	// WX2A ROT
IF WX2TargetPos.nRotPos + WX2TargetPos.nRotCatch > WX^.Rot_A.Out.DistancePos_PO AND
	WX2TargetPos.nRotPos - WX2TargetPos.nRotCatch < WX^.Rot_A.Out.DistancePos_PO THEN
		WX^.Rot_A.bStopMove := TRUE;
END_IF

	// WX2A CLAMP
IF WX2TargetPos.nClampPos + WX2TargetPos.nClampCatch > WX^.Clamp_A.Out.DistancePos_PO AND
	WX2TargetPos.nClampPos - WX2TargetPos.nClampCatch < WX^.Clamp_A.Out.DistancePos_PO THEN
		WX^.Clamp_A.bStopMove := TRUE;
END_IF

	// WX2B VERT
IF WX2TargetPos.nVertPos + WX2TargetPos.nVertCatch > WX^.Vert_B.Out.DistancePos_PO AND
	WX2TargetPos.nVertPos - WX2TargetPos.nVertCatch < WX^.Vert_B.Out.DistancePos_PO THEN
		WX^.Vert_B.bStopMove := TRUE;
END_IF

	// WX2B ROT
IF WX2TargetPos.nRotPos + WX2TargetPos.nRotCatch > WX^.Rot_B.Out.DistancePos_PO AND
	WX2TargetPos.nRotPos - WX2TargetPos.nRotCatch < WX^.Rot_B.Out.DistancePos_PO THEN
		WX^.Rot_B.bStopMove := TRUE;
END_IF

	// WX2B CLAMP
IF WX2TargetPos.nClampPos + WX2TargetPos.nClampCatch > WX^.Clamp_B.Out.DistancePos_PO AND
	WX2TargetPos.nClampPos - WX2TargetPos.nClampCatch < WX^.Clamp_B.Out.DistancePos_PO THEN
		WX^.Clamp_B.bStopMove := TRUE;
END_IF




	// This is to give the axes time to stop, before we move onto the next step
IF WX^.Vert_A.StopCase = 100 AND WX^.Rot_A.StopCase = 100 AND WX^.Clamp_A.StopCase = 100 AND
	WX^.Vert_B.StopCase = 100 AND WX^.Rot_B.StopCase = 100 AND WX^.Clamp_B.StopCase = 100 THEN
	bInPosition := TRUE;
ELSE
	bInPosition := FALSE;
END_IF

IF bClamped THEN
	IF WX^.Vert_A.StopCase = 100 AND WX^.Rot_A.StopCase = 100 AND WX^.Vert_B.StopCase = 100 THEN
		bInPosition := TRUE;
	ELSE
		bInPosition := FALSE;
	END_IF
END_IF

armsInTargetPosition := bInPosition;
END_METHOD

METHOD CleanUpMove : BOOL
(*
	This method assumes that the movement from the initial 'big' move has ended.
*)
IF NOT bInitCleanUpTrigger THEN
	enableAltSpeed();
	
		// Reload Target Position into our ClearpathPositionABS
	WX^.VertDisReq_PI 	:= REAL_TO_INT(WX2TargetPos.nVertPos);
	WX^.RotDegReq_PI  	:= REAL_TO_INT(WX2TargetPos.nRotPos);
	WX^.ClampDisReq_PI := REAL_TO_INT(WX2TargetPos.nClampPos);
	
		// If we are clamped, we don't move all axis
	IF NOT bClamped THEN
		WX^.bPresetMoveTrigger := TRUE;
	ELSE
		WX^.Vert_A.bPresetMoveTrigger := TRUE;
		WX^.Vert_B.bPresetMoveTrigger := TRUE;
		WX^.Rot_A.bPresetMoveTrigger  := TRUE;
			
		WX^.Vert_A.bMove_PI := TRUE;
		WX^.Vert_B.bMove_PI := TRUE;
		WX^.Rot_A.bMove_PI  := TRUE;
	END_IF
	
	enableAltSpeed();
	
	bInitCleanUpTrigger     := TRUE;
END_IF

enableAltSpeed();

CleanUpMove := precisionMoveChecker();
END_METHOD

METHOD disableAltSpeed : BOOL
VAR
	bDetect : BOOL := FALSE;
END_VAR

(* 
	This method returns TRUE if  alt speed control was DISABLED already.
*)
bDetect := FALSE;

IF NOT WX^.Vert_A.bAltSpeedControl OR NOT WX^.Vert_B.bAltSpeedControl  THEN
	bDetect := TRUE;
END_IF

IF NOT WX^.Rot_A.bAltSpeedControl OR NOT WX^.Rot_B.bAltSpeedControl THEN
	bDetect := TRUE;
END_IF

IF NOT WX^.Clamp_A.bAltSpeedControl OR NOT WX^.Clamp_A.bAltSpeedControl THEN
	bDetect := TRUE;
END_IF

WX^. Vert_A.bAltSpeedControl := FALSE;
WX^.  Rot_A.bAltSpeedControl := FALSE;
WX^.Clamp_A.bAltSpeedControl := FALSE;

WX^. Vert_B.bAltSpeedControl := FALSE;
WX^.  Rot_B.bAltSpeedControl := FALSE;
WX^.Clamp_A.bAltSpeedControl := FALSE;

disableAltSpeed := bDetect;
END_METHOD

METHOD enableAltSpeed : BOOL
VAR
	bDetect : BOOL := FALSE;
END_VAR
(* 
	This method returns TRUE if  alt speed control was ENABLED already.
*)
bDetect := FALSE;

IF WX^.Vert_A.bAltSpeedControl OR WX^.Vert_B.bAltSpeedControl  THEN
	bDetect := TRUE;
END_IF

IF WX^.Rot_A.bAltSpeedControl OR WX^. Rot_B.bAltSpeedControl THEN
	bDetect := TRUE;
END_IF

IF WX^.Clamp_A.bAltSpeedControl OR WX^.Clamp_B.bAltSpeedControl THEN
	bDetect := TRUE;
END_IF

WX^. Vert_A.bAltSpeedControl := TRUE;
WX^.  Rot_A.bAltSpeedControl := TRUE;
WX^.Clamp_A.bAltSpeedControl := TRUE;

WX^. Vert_B.bAltSpeedControl := TRUE;
WX^.  Rot_B.bAltSpeedControl := TRUE;
WX^.Clamp_B.bAltSpeedControl := TRUE;

enableAltSpeed := bDetect;
END_METHOD

METHOD MoveArms : BOOL
VAR_INPUT
	position : sBogieArmPosition;
END_VAR
(*
	Author @ Joseph Barton	

	This method is initiating and monitoring the initial move for a preset move command.
*)

	// If we are not busy moving somewhere.
IF NOT bBusy THEN	
	bBusy 		  := TRUE;	// We are now busy.
	bMoveComplete := FALSE;	// And our move is not complete.
							// 	If we are already in the target position,
							// 	That will be determined later in this cycle.
	tStartTime := TIME(); 	// Save the start time, for the timeout error tracking.
							
		// This is the 'big' move, so we disable altenate speed to move quickly
	disableAltSpeed();		
	
		// set our target position for position checking.
	WX2TargetPos := position;	
	
		// Tell the Auto-movement part of our clearpath library our desired location.
	WX^.VertDisReq_PI 	:= REAL_TO_INT(WX2TargetPos.nVertPos); 	
	WX^.RotDegReq_PI  	:= REAL_TO_INT(WX2TargetPos.nRotPos);
	WX^.ClampDisReq_PI := REAL_TO_INT(WX2TargetPos.nClampPos);
	
		// IF we are NOT clamped we can use the bPresetMoveTrigger boolean to
		//		give the library the right information on how te move.
	IF NOT bClamped THEN
		WX^.bPresetMoveTrigger := TRUE;
	ELSE
		
			// If we are clamped, then we cannot move all 6 motors,
			//		and we have to manually tell our desired axis
			//		that we are moving them to a preset position.
		WX^.Vert_A.bPresetMoveTrigger := TRUE;
		WX^.Vert_B.bPresetMoveTrigger := TRUE;
		WX^.Rot_A.bPresetMoveTrigger  := TRUE;
		
			// Then tell them to move.
		WX^.Vert_A.bMove_PI := TRUE;
		WX^.Vert_B.bMove_PI := TRUE;
		WX^.Rot_A.bMove_PI  := TRUE;
	END_IF
	
	disableAltSpeed();
END_IF

	// disableing alternate speed each cycle is too much,
	//		but there is a glitch where it will go into
	// 		alternate speed 'randomly'. I will have to
	//		fix it soon.
disableAltSpeed();

	// Check if we are in the correct position each cycle.
MoveArms := armsInTargetPosition();
END_METHOD

METHOD partPresent : BOOL
VAR_INPUT
END_VAR

(* 
	This method returns true if there is a part detected by the part present sensor.
	
	This still needs to be implemented, but because the Part Present Sensors do not exist yet, this is what we got.
*)
partPresent := FALSE;
END_METHOD

METHOD precisionMoveChecker : BOOL
VAR
	bWX2AVertInLocation  : BOOL := FALSE;
	bWX2ARotInLocation   : BOOL := FALSE;
	bWX2AClampInLocation : BOOL := FALSE;
	
	bWX2BVertInLocation  : BOOL := FALSE;
	bWX2BRotInLocation 	 : BOOL := FALSE;
	bWX2BClampInLocation : BOOL := FALSE;
END_VAR
	// Vert_A
IF WX2TargetPos.nVertPos + WX2TargetPos.nVertTolerance > WX^.Vert_A.Out.DistancePos_PO AND
 	WX2TargetPos.nVertPos - WX2TargetPos.nVertTolerance < WX^.Vert_A.Out.DistancePos_PO THEN
		bWX2AVertInLocation := TRUE;
		WX^.Vert_A.bStopMove := TRUE;
ELSE
	WX^.Vert_A.bStopMove := FALSE;
END_IF
	
	// Rot_A
IF WX2TargetPos.nRotPos + WX2TargetPos.nRotTolerance > WX^.Rot_A.Out.DistancePos_PO AND
	WX2TargetPos.nRotPos - WX2TargetPos.nRotTolerance < WX^.Rot_A.Out.DistancePos_PO THEN
		bWX2ARotInLocation := TRUE;
		WX^.Rot_A.bStopMove := TRUE;
ELSE
	WX^.Rot_A.bStopMove := FALSE;
END_IF

	// Clamp_A
IF WX2TargetPos.nClampPos + WX2TargetPos.nClampTolerance > WX^.Clamp_A.Out.DistancePos_PO AND
	WX2TargetPos.nClampPos - WX2TargetPos.nClampTolerance < WX^.Clamp_A.Out.DistancePos_PO THEN
		bWX2AClampInLocation := TRUE;
		WX^.Clamp_A.bStopMove := TRUE;
ELSE
	WX^.Clamp_A.bStopMove := FALSE;
END_IF

	// Vert_B
IF WX2TargetPos.nVertPos + WX2TargetPos.nVertTolerance > WX^.Vert_B.Out.DistancePos_PO AND
 	WX2TargetPos.nVertPos - WX2TargetPos.nVertTolerance < WX^.Vert_B.Out.DistancePos_PO THEN
		bWX2BVertInLocation := TRUE;
		WX^.Vert_B.bStopMove := TRUE;
ELSE
	WX^.Vert_B.bStopMove := FALSE;
END_IF
	
	// Rot_B
IF WX2TargetPos.nRotPos + WX2TargetPos.nRotTolerance > WX^.Rot_B.Out.DistancePos_PO AND
	WX2TargetPos.nRotPos - WX2TargetPos.nRotTolerance < WX^.Rot_B.Out.DistancePos_PO THEN
		bWX2BRotInLocation := TRUE;
		WX^.Rot_B.bStopMove := TRUE;
ELSE
	WX^.Rot_B.bStopMove := FALSE;
END_IF

	// Clamp_B
IF WX2TargetPos.nClampPos + WX2TargetPos.nClampTolerance > WX^.Clamp_B.Out.DistancePos_PO AND
	WX2TargetPos.nClampPos - WX2TargetPos.nClampTolerance < WX^.Clamp_B.Out.DistancePos_PO THEN
		bWX2BClampInLocation := TRUE;
		WX^.Clamp_B.bStopMove := TRUE;
ELSE
	WX^.Clamp_B.bStopMove := FALSE;
END_IF

	// Check if all axis are in location, and return TRUE; ELSE return FALSE;
IF bWX2AVertInLocation AND bWX2ARotInLocation AND bWX2AClampInLocation AND
	bWX2BVertInLocation AND bWX2BRotInLocation AND bWX2BClampInLocation THEN
		
		WX^.Clamp_B.bStopMove := FALSE;
		WX^.Rot_B.bStopMove := FALSE;
		WX^.Vert_B.bStopMove := FALSE;
		WX^.Clamp_A.bStopMove := FALSE;
		WX^.Rot_A.bStopMove := FALSE;
		WX^.Vert_A.bStopMove := FALSE;
		
		precisionMoveChecker := TRUE;
	
ELSE
	precisionMoveChecker := FALSE;
END_IF

	// IF we are clamped then we are checking for the Vert_A, Vert_B, & Rot_A axis only.
IF bClamped THEN
	IF bWX2AVertInLocation AND bWX2ARotInLocation AND bWX2BVertInLocation THEN
		
		WX^.Vert_B.bStopMove := FALSE;
		WX^.Rot_A.bStopMove := FALSE;
		WX^.Vert_A.bStopMove := FALSE;
		
		precisionMoveChecker := TRUE;
	END_IF
END_IF
END_METHOD

ACTION startAllMovement:
WX^.Vert_A.bStopMove 	:= FALSE;
WX^.Rot_A.bStopMove 	:= FALSE;
WX^.Clamp_A.bStopMove 	:= FALSE;
WX^.Vert_B.bStopMove 	:= FALSE;
WX^.Rot_B.bStopMove  	:= FALSE;
WX^.Clamp_B.bStopMove 	:= FALSE;
END_ACTION

ACTION stopAllMovement:
WX^.Vert_A.bStopMove 	:= TRUE;
WX^.Rot_A.bStopMove 	:= TRUE;
WX^.Clamp_A.bStopMove 	:= TRUE;
WX^.Vert_B.bStopMove 	:= TRUE;
WX^.Rot_B.bStopMove 	:= TRUE;
WX^.Clamp_B.bStopMove 	:= TRUE;
END_ACTION

END_FUNCTION_BLOCK

// ---- Machine System/FUNCTIONS/F_PartIsPresent.TcPOU
FUNCTION F_PartIsPresent : BOOL
VAR_INPUT
	WX : sBogie;
END_VAR
VAR
END_VAR

IF (WX.A.bPP1_Input AND WX.A.bPP2_Input AND WX.B.bPP1_Input AND WX.A.bPP2_Input) OR NOT(WX.bEnabled) THEN
	F_PartIsPresent := 1;
	ELSE
		F_PartIsPresent := 0;
END_IF

END_FUNCTION

// ---- Machine System/FUNCTIONS/F_PartIsPresentAndClamped.TcPOU
FUNCTION F_PartIsPresentAndClamped : BOOL
VAR_INPUT
	WX : sBogie;
END_VAR
VAR
END_VAR

IF (WX.A.bPP1_Input AND WX.A.bPP2_Input AND WX.B.bPP1_Input AND WX.A.bPP2_Input AND WX.A.bClamped AND WX.B.bClamped) OR NOT(WX.bEnabled) THEN
	F_PartIsPresentAndClamped := 1;
	ELSE
		F_PartIsPresentAndClamped := 0;
END_IF

END_FUNCTION

// ---- Machine System/FUNCTIONS/F_IsEmpty.TcPOU
FUNCTION F_IsEmpty : BOOL
VAR_INPUT
	WX : sBogie;
END_VAR
VAR
END_VAR

IF WX.A.bPP1_Input = 0 AND WX.A.bPP2_Input = 0 AND WX.B.bPP2_Input = 0 AND WX.B.bPP2_Input = 0 THEN
	F_IsEmpty := 1;
	ELSE 
		F_IsEmpty := 0;
END_IF

END_FUNCTION

// ---- Machine System/FUNCTIONS/F_ArmsInLoadOrientation.TcPOU
FUNCTION F_ArmsInLoadOrientation : BOOL
VAR_INPUT
END_VAR
VAR
END_VAR

END_FUNCTION

// ---- Machine System/FUNCTIONS/F_PartPickupSuccess.TcPOU
FUNCTION F_PartPickupSuccess : BOOL
VAR_INPUT
	WX : sBogie;
END_VAR
VAR
END_VAR

IF WX.bEnabled THEN
	IF WX.A.bClamped AND WX.B.bClamped AND F_PartIsPresent(WX) AND WX.ConveyorLoadPos = 0 THEN
		
		F_PartPickupSuccess := 1;
 
	ELSE
		F_PartPickupSuccess := 0;
		RETURN;
	END_IF
	
	RETURN;
	
END_IF

END_FUNCTION

// ---- Machine System/FUNCTIONS/F_CheckMoldData.TcPOU
FUNCTION F_CheckMoldData : BOOL
VAR_INPUT
	MoldID 		: INT;
	WX_Enable	: BOOL;
END_VAR
VAR
END_VAR

//Function to check the database for each file string and check for the file on the system 
IF WX_Enable THEN
	IF MoldID = 0 THEN
		RETURN;
		ELSE
			F_CheckMoldData := 1;
		END_IF
	ELSE
		F_CheckMoldData := 1;
END_IF

END_FUNCTION

// ---- CNC HMI/CNC_HMI_HLI_Added_Code.TcPOU
PROGRAM CNC_HMI_HLI_Added_Code
VAR
Scaler : INT :=10000; //change to a scaling variable when deciding to use inches
mdiTest : STRING;
//EventLogger page Reset
	fbEventlogger : FB_TcEventLogger;
	fbAlarm: FB_TcAlarm;
	fbMessage: FB_TcMessage;
	bAlarm: BOOL;
	bMessage : BOOL;
	bIsInitalized: BOOL;
	bClearAlarm: BOOL;
	bConfirmAlarm: BOOL;
//ch1
	SP1_X : fb_HMI_AX;
	SP1_Y : fb_HMI_AX;
	SP1_Z : fb_HMI_AX;
	SP1_A : fb_HMI_AX;
	SP1_C : fb_HMI_AX;
//ch2
	R1_X	: fb_HMI_AX;
	R1_Y	: fb_HMI_AX;
	R1_Z1	: fb_HMI_AX;
	R1_Z2	: fb_HMI_AX;
	R1_C	: fb_HMI_AX;
	
//axis1
(*
Spray_Axis1 : STRING;
SP1_PCS		: STRING;
SP1_ACS		: STRING;
SP1_cmd		: STRING;
SP1_Min		: STRING;
SP1_Max		: STRING;
//axis2

Spray_Axis2 : STRING;
SP2_PCS		: STRING;
SP2_ACS		: STRING;
SP2_cmd		: STRING;
SP2_Min		: STRING;
SP2_Max		: STRING;
SP2_Feed	: string;
//axis3
Spray_Axis3 : STRING;
SP3_PCS		: STRING;
SP3_ACS		: STRING;
SP3_cmd		: STRING;
SP3_min		: STRING;
SP3_max		: STRING;
//axis4
Spray_Axis4 : STRING;
SP4_PCS		: STRING;
SP4_ACS		: STRING;
SP4_cmd		: STRING;
SP4_min		: STRING;
SP4_max		: STRING;
//axis5
Spray_Axis5 : STRING;
SP5_PCS		: STRING;
SP5_ACS		: STRING;
SP5_cmd		: STRING;
Sp5_min		: STRING;
SP5_Max		: STRING;

//channel 2
//axis1
Roll_Axis1 	: STRING;
R1_PCS		: STRING;
R1_ACS		: STRING;
R1_cmd		: STRING;
R1_Min		: STRING;
R1_Max		: STRING;
//axis2
Roll_Axis2 	: STRING;
R2_PCS		: STRING;
R2_ACS		: STRING;
R2_cmd		: STRING;
//axis3
Roll_Axis3 	: STRING;
R3_PCS		: STRING;
R3_ACS		: STRING;
R3_cmd		: STRING;
//axis4
Roll_Axis4 	: STRING;
R4_PCS		: STRING;
R4_ACS		: STRING;
R4_cmd		: STRING;
//axis5
Roll_Axis5 	: STRING;
R5_PCS		: STRING;
R5_ACS		: STRING;
R5_cmd		: STRING;
//axis6
Roll_Axis6 	: STRING;
R6_PCS		: STRING;
R6_ACS		: STRING;
R6_cmd		: STRING;
*)
//gcode access See PRG 'P_GFuctionMonitor()'

END_VAR


// read gcode buffer
	P_GFunctionMonitor();	//Channel 1 G Code Reader
	//P_GFunctionMonitor_2(); 	//channel 2 G Code Reader
//EventLogger Buttons for reset
//	IF NOT bIsInitalized THEN
//	bIsInitalized := TRUE;
//	fbMessage.CreateEx(TC_Events.MyEvents.Start, 0);
//	fbAlarm.CreateEx(TC_Events.MyEvents.Stop, TRUE, 0);
//	END_IF
//	//Test git
//	IF bMessage THEN
//		bMessage := FALSE;
//		fbMessage.Send(0);
//	END_IF
	
//	IF bAlarm THEN
//		bAlarm := FALSE;
//		fbAlarm.Raise(0);
//	END_IF
	
//	IF bClearAlarm THEN
//		bClearAlarm := FALSE;
//		fbAlarm.Clear(0, TRUE);
//	END_IF
//ch1 fb
	SP1_X(chId:=0,chAx:=0,Scaler:=Scaler);
	SP1_Y(chId:=0,chAx:=1,Scaler:=Scaler);
	SP1_Z(chId:=0,chAx:=2,Scaler:=Scaler);
	SP1_A(chId:=0,chAx:=3,Scaler:=Scaler);
	SP1_C(chId:=0,chAx:=4,Scaler:=Scaler);
//ch2 fb
	R1_X(chId:=1,chAx:=0,Scaler:=Scaler);
	R1_Y(chId:=1,chAx:=1,Scaler:=Scaler);
	R1_Z1(chId:=1,chAx:=2,Scaler:=Scaler);
	R1_Z2(chId:=1,chAx:=3,Scaler:=Scaler);
	R1_C(chId:=1,chAx:=4,Scaler:=Scaler);
	
(*  Method for HMI before FB was added.  Use this if While loop fails
	Spray_Axis1 := gpCh[0]^.bahn_state.coord_r[0].axis_name_r.zeichen;
	SP1_PCS		:= FLOAT_TO_STRING(Dint_to_float(gpCh[0]^.bahn_state.coord_r[0].current_position_r)/Scaler);
	SP1_ACS		:= FLOAT_TO_STRING(Dint_to_float(gpCh[0]^.bahn_state.coord_r[0].acs_position_r)/Scaler);
	SP1_CMD		:= FLOAT_TO_STRING(DINT_TO_FLOAT(gpCh[0]^.bahn_state.coord_r[0].cmd_position_r)/Scaler);
	SP1_Min 	:= FLOAT_TO_STRING(DINT_TO_FLOAT(gpAx[0]^.lr_state.conf_neg_software_limit_r)/Scaler);
	SP1_Max 	:= FLOAT_TO_STRING(DINT_TO_FLOAT(gpAx[0]^.lr_state.conf_pos_software_limit_r)/Scaler);
	Spray_Axis2 := gpCh[0]^.bahn_state.coord_r[1].axis_name_r.zeichen;
	SP2_PCS		:= FLOAT_TO_STRING(Dint_to_float(gpCh[0]^.bahn_state.coord_r[1].current_position_r)/Scaler);
	SP2_ACS		:= FLOAT_TO_STRING(Dint_to_float(gpCh[0]^.bahn_state.coord_r[1].acs_position_r)/Scaler);
	SP2_CMD		:= FLOAT_TO_STRING(DINT_TO_FLOAT(gpCh[0]^.bahn_state.coord_r[1].cmd_position_r)/Scaler);
	SP2_Min 	:= FLOAT_TO_STRING(DINT_TO_FLOAT(gpAx[1]^.lr_state.conf_neg_software_limit_r)/Scaler);
	SP2_Max 	:= FLOAT_TO_STRING(DINT_TO_FLOAT(gpAx[1]^.lr_state.conf_pos_software_limit_r)/Scaler);
	SP2_Feed	:= DINT_TO_STRING(gpch[0]^.bahn_state.coord_r[1].w0_velocity_r);
	
	Spray_Axis3 := gpCh[0]^.bahn_state.coord_r[2].axis_name_r.zeichen;
	SP3_PCS		:= FLOAT_TO_STRING(Dint_to_float(gpCh[0]^.bahn_state.coord_r[2].current_position_r)/Scaler);
	SP3_ACS		:= FLOAT_TO_STRING(Dint_to_float(gpCh[0]^.bahn_state.coord_r[2].acs_position_r)/Scaler);
	SP3_CMD		:= FLOAT_TO_STRING(DINT_TO_FLOAT(gpCh[0]^.bahn_state.coord_r[2].cmd_position_r)/Scaler);
	SP3_Min 	:= FLOAT_TO_STRING(DINT_TO_FLOAT(gpAx[2]^.lr_state.conf_neg_software_limit_r)/Scaler);
	SP3_Max 	:= FLOAT_TO_STRING(DINT_TO_FLOAT(gpAx[2]^.lr_state.conf_pos_software_limit_r)/Scaler);
	
	Spray_Axis4 := gpCh[0]^.bahn_state.coord_r[3].axis_name_r.zeichen;
	SP4_PCS		:= FLOAT_TO_STRING(Dint_to_float(gpCh[0]^.bahn_state.coord_r[3].current_position_r)/Scaler);
	SP4_ACS		:= FLOAT_TO_STRING(Dint_to_float(gpCh[0]^.bahn_state.coord_r[3].acs_position_r)/Scaler);
	SP4_CMD		:= FLOAT_TO_STRING(DINT_TO_FLOAT(gpCh[0]^.bahn_state.coord_r[3].cmd_position_r)/Scaler);
	SP4_Min 	:= FLOAT_TO_STRING(DINT_TO_FLOAT(gpAx[3]^.lr_state.conf_neg_software_limit_r)/Scaler);
	SP4_Max 	:= FLOAT_TO_STRING(DINT_TO_FLOAT(gpAx[3]^.lr_state.conf_pos_software_limit_r)/Scaler);
	
	Spray_Axis5 := gpCh[0]^.bahn_state.coord_r[4].axis_name_r.zeichen;
	SP5_PCS		:= FLOAT_TO_STRING(Dint_to_float(gpCh[0]^.bahn_state.coord_r[4].current_position_r)/Scaler);
	SP5_ACS		:= FLOAT_TO_STRING(Dint_to_float(gpCh[0]^.bahn_state.coord_r[4].acs_position_r)/Scaler);
	SP5_CMD		:= FLOAT_TO_STRING(DINT_TO_FLOAT(gpCh[0]^.bahn_state.coord_r[4].cmd_position_r)/Scaler);
	SP5_Min 	:= FLOAT_TO_STRING(DINT_TO_FLOAT(gpAx[4]^.lr_state.conf_neg_software_limit_r)/Scaler);
	SP5_Max 	:= FLOAT_TO_STRING(DINT_TO_FLOAT(gpAx[4]^.lr_state.conf_pos_software_limit_r)/Scaler);
	
	//channel2
	Roll_Axis1 	:= gpCh[1]^.bahn_state.coord_r[0].axis_name_r.zeichen;
	R1_PCS		:= FLOAT_TO_STRING(Dint_to_float(gpCh[1]^.bahn_state.coord_r[0].current_position_r)/Scaler);
	R1_ACS		:= FLOAT_TO_STRING(Dint_to_float(gpCh[1]^.bahn_state.coord_r[0].acs_position_r)/Scaler);
	R1_CMD		:= FLOAT_TO_STRING(Dint_to_float(gpCh[1]^.bahn_state.coord_r[0].cmd_position_r)/Scaler);
	R1_Min 		:= FLOAT_TO_STRING(DINT_TO_FLOAT(gpAx[0]^.lr_state.conf_neg_software_limit_r)/Scaler);
	R1_Max 		:= FLOAT_TO_STRING(DINT_TO_FLOAT(gpAx[0]^.lr_state.conf_pos_software_limit_r)/Scaler);
	
	Roll_Axis2 	:= gpCh[1]^.bahn_state.coord_r[1].axis_name_r.zeichen;
	R2_PCS		:= FLOAT_TO_STRING(Dint_to_float(gpCh[1]^.bahn_state.coord_r[1].current_position_r)/Scaler);
	R2_ACS		:= FLOAT_TO_STRING(Dint_to_float(gpCh[1]^.bahn_state.coord_r[1].acs_position_r)/Scaler);
	R2_CMD		:= FLOAT_TO_STRING(Dint_to_float(gpCh[1]^.bahn_state.coord_r[1].cmd_position_r)/Scaler);
	
	Roll_Axis3 := gpCh[1]^.bahn_state.coord_r[2].axis_name_r.zeichen;
	R3_PCS		:= FLOAT_TO_STRING(Dint_to_float(gpCh[1]^.bahn_state.coord_r[2].current_position_r)/Scaler);
	R3_ACS		:= FLOAT_TO_STRING(Dint_to_float(gpCh[1]^.bahn_state.coord_r[2].acs_position_r)/Scaler);
	R3_CMD		:= FLOAT_TO_STRING(Dint_to_float(gpCh[1]^.bahn_state.coord_r[2].cmd_position_r)/Scaler);
	
	Roll_Axis4 := gpCh[1]^.bahn_state.coord_r[3].axis_name_r.zeichen;
	R4_PCS		:= FLOAT_TO_STRING(Dint_to_float(gpCh[1]^.bahn_state.coord_r[3].current_position_r)/Scaler);
	R4_ACS		:= FLOAT_TO_STRING(Dint_to_float(gpCh[1]^.bahn_state.coord_r[3].acs_position_r)/Scaler);
	R4_CMD		:= FLOAT_TO_STRING(Dint_to_float(gpCh[1]^.bahn_state.coord_r[3].cmd_position_r)/Scaler);
	
	Roll_Axis5 := gpCh[1]^.bahn_state.coord_r[4].axis_name_r.zeichen;
	R5_PCS		:= FLOAT_TO_STRING(Dint_to_float(gpCh[1]^.bahn_state.coord_r[4].current_position_r)/Scaler);
	R5_ACS		:= FLOAT_TO_STRING(Dint_to_float(gpCh[1]^.bahn_state.coord_r[4].acs_position_r)/Scaler);
	R5_CMD		:= FLOAT_TO_STRING(Dint_to_float(gpCh[1]^.bahn_state.coord_r[4].cmd_position_r)/Scaler);
	
	Roll_Axis6 := gpCh[1]^.bahn_state.coord_r[5].axis_name_r.zeichen;
	R6_PCS		:= FLOAT_TO_STRING(Dint_to_float(gpCh[1]^.bahn_state.coord_r[5].current_position_r)/Scaler);
	R6_ACS		:= FLOAT_TO_STRING(Dint_to_float(gpCh[1]^.bahn_state.coord_r[5].acs_position_r)/Scaler);
	R6_CMD		:= FLOAT_TO_STRING(Dint_to_float(gpCh[1]^.bahn_state.coord_r[5].cmd_position_r)/Scaler);
*)

END_PROGRAM

// ---- CNC HMI/fb_HMI_AX.TcPOU
FUNCTION_BLOCK fb_HMI_AX
VAR_INPUT
	chId	: INT;	//channel id from cnc configuration
	chAx	: INT;	//default index setting in cnc channel config
	Scaler	: INT;	//scaler used to move from micro mm to mm (can also be changed in plc to get to inches)
	viSelectAx : BOOL; //select this axis on hmi
END_VAR
VAR_OUTPUT
	Name 	: STRING;
	PCS 	: STRING;
	ACS		: LReal;
	CMD		: STRING;
	PosMin	: LREAL;
	PosMax	: LREAL;
	manualActive : BOOL;
	selectedAx : INT;
	Feed : STRING;
	Feed2 : STRING;
	Feed3 : STRING;
	tf1 : LREAL;
	tf2 : LREAL;
	tf3 : LREAL;
	tf4 : STRING;
	tf5 : string;
	//Feed4 : string;
END_VAR
VAR
	axID		: UINT;
	axLogN		:UINT;
	chLogN		:UINT;
	m			: int;
END_VAR

//Idea of this fb is to create a scalable method to display axis data on the new twincat hmi display no matter how many axis get added to a channel
chLogN	:= gpCh[chId]^.bahn_state.coord_r[chAx].log_achs_nr_r; //this is located in motion paramters when adding axis to project
axLogN 	:= gpAx[m]^.head.log_ax_nr_r;
WHILE chLogN <> axLogN AND m<255 DO //m<255
	m := m+1;
	axLogN 	:= gpAx[m]^.head.log_ax_nr_r;
END_WHILE

Name 	 := gpCh[chId]^.bahn_state.coord_r[chAx].axis_name_r.zeichen;
PCS		 := FLOAT_TO_STRING(Dint_to_float(gpCh[chId]^.bahn_state.coord_r[chAx].current_position_r)/Scaler);
ACS		 := (Dint_to_float(gpCh[chid]^.bahn_state.coord_r[chAx].acs_position_r)/Scaler);
CMD		 := FLOAT_TO_STRING(DINT_TO_FLOAT(gpCh[chid]^.bahn_state.coord_r[chAx].cmd_position_r)/Scaler);
PosMin	 := (DINT_TO_FLOAT(gpAx[m]^.lr_state.conf_neg_software_limit_r)/Scaler);
PosMax	 := (DINT_TO_FLOAT(gpAx[m]^.lr_state.conf_pos_software_limit_r)/Scaler);
tf1	 := (DINT_TO_FLOAT(gpAx[m]^.lr_state.current_rev_r)/Scaler);
tf2	 := (Dint_to_float(gpCh[chid]^.bahn_state.active_feed_r)/Scaler);
//tf3	 := GVL_Machine.pCh0^.bahn_state.coord_r[2].w0_velocity_r;
tf3	 := gpCh[chId]^.bahn_state.coord_r[chAx].w0_velocity_r;
//Feed 	 := Float_to_string(Dint_to_Float(gpCH[chId]^.bahn_state.active_feed_r)/Scaler);
//Feed2 	 := Float_to_string(Dint_to_Float(gpCH[chId]^.bahn_state.command_feed_r)/Scaler);
//Feed3 	 := Float_to_string(Dint_to_Float(gpCH[chId]^.bahn_state.command_feed_active_r)/Scaler);
////Feed4 	 := Float_to_string(Dint_to_Float(gpCH[chId]^.bahn_state.coord_r)/Scaler);


IF global_hmi.PLCMachineMode[chID].ManualMode.nLogAxisNumber = axLogN THEN
	manualActive := TRUE;
	else manualActive :=false;
END_IF
IF viSelectAx THEN
	global_hmi.PLCMachineMode[chID].ManualMode.nLogAxisNumber := axLogN;
	viSelectAx := false;
END_IF

END_FUNCTION_BLOCK

// ---- CNC HMI/P_GFunctionMonitor.TcPOU
PROGRAM P_GFunctionMonitor
VAR
	rtM100 :r_trig;
	ch1_actM_r : STRING;
	mcode1 : BOOL;
	mcode2: BOOL;
	mcode3: bool;
	bReadGcode: BOOL;
	fbADSRead: ADSREADEX;
	GBuffer: ARRAY[1..39]OF WORD;
	nPathPrep: WORD;
	nPlane: WORD;
	nCutterComp: WORD;
	nDeselectDiamProg: WORD;
	nZeroOffset: WORD;
	nContMode: WORD;
	nMeasureMode: WORD;
	nDeselectSpline: WORD;
	nDeselectCornerRed: WORD;
	//toString
		sPathPrep: STRING;
		sPlane: STRING;
		sCutterComp: STRING;
		sDeselectDiamProg: STRING;
		sZeroOffset: STRING;
		sContMode: STRING;
		sMeasureMode: STRING;
		sDeselectSpline: STRING;
		sDeselectCornerRed: STRING;
	fbUpdate: TON;
	sLocalAmsNet 	: STRING; 
	getAmsNet : FB_GetLocalAmsNetId;
	bLocalAmsNet : BOOL;
	
	sGCodeOut : string;
END_VAR


//Read active G code
IF sLocalAmsNet ='' THEN
	bLocalAmsNet := TRUE;
ELSE
	blocalamsNet := FALSE;
END_IF
getAmsNet(bExecute:=bLocalAmsNet, tTimeOut:=DEFAULT_ADS_TIMEOUT,AddrString => sLocalAmsNet);

IF Global_HMI.PLCSelectedChannel = 0 THEN
	bReadGcode := TRUE;
	ELSE breadgcode := FALSE;
END_IF
fbUpdate.PT := T#1S;
IF bReadGcode THEN
	fbUpdate.IN := TRUE;
ELSE
	fbUpdate.IN := FALSE;
END_IF

IF fbUpdate.Q THEN
	fbADSRead(
	NETID:=sLocalAmsNet, 
	PORT:=553, 
	IDXGRP:=16#120101, 
	IDXOFFS:=16#3C, 
	LEN:=SIZEOF(GBuffer), 
	DESTADDR:=ADR(GBuffer), 
	READ:=TRUE, 
	TMOUT:=T#2S, 
	BUSY=> , 
	ERR=> , 
	ERRID=> , 
	COUNT_R=> );
	
	IF NOT fbADSRead.BUSY THEN
		fbADSRead(
			NETID:=sLocalAmsNet, 
			PORT:=553, 
			IDXGRP:=16#120101, 
			IDXOFFS:=16#3C, 
			LEN:=SIZEOF(GBuffer), 
			DESTADDR:=ADR(GBuffer), 
			READ:=FALSE, 
			TMOUT:=T#2S);
		fbUpdate.IN := FALSE;
	END_IF
END_IF
//Parse them out
nPathPrep 			:= GBuffer[1];
nPlane 				:= GBuffer[5];
nCutterComp 		:= GBuffer[8];
nDeselectDiamProg 	:= GBuffer[9];
nZeroOffset 		:= GBuffer[10];
nContMode			:= GBuffer[11];
nMeasureMode 		:= GBuffer[15];
nDeselectSpline 	:= GBuffer[30];
nDeselectCornerRed 	:= GBuffer[32];
//to string
IF 	nPathPrep > 0 AND npathprep< 65535 THEN
	sPathPrep:= concat(concat('G',TO_STRING(nPathPrep)),' '); ELSE sPathPrep :=''; END_IF
IF nPlane >0 AND nPlane<65535 THEN
	sPlane:= concat(concat('G',TO_STRING(nPlane)),' '); ELSE sPlane:=''; END_IF
IF nCutterComp>0 AND nCutterComp<65535 THEN
	sCutterComp:= concat(concat('G',TO_STRING(nCutterComp)),' '); ELSE sCutterComp :=''; END_IF
IF nDeselectDiamProg >0 AND nDeselectDiamProg<65535 THEN
	sDeselectDiamProg:= concat(concat('G',TO_STRING(nDeselectDiamProg)),' '); ELSE sDeselectDiamProg :=''; END_IF
IF nZeroOffset >0 AND nZeroOffset<65535 THEN
	sZeroOffset:= concat(concat('G',TO_STRING(nZeroOffset)),' '); ELSE sZeroOffset:=''; END_IF
IF ncontmode > 0 AND ncontmode < 65535 THEN
	sContMode:= concat(concat('G',TO_STRING(nContMode)),' '); ELSE scontmode:=''; END_IF
IF nMeasureMode >0 AND nMeasureMode < 65535 THEN
	sMeasureMode:= concat(concat('G',TO_STRING(nMeasureMode)),' '); ELSE sMeasureMode := ''; END_IF
IF 	nDeselectSpline > 0 AND nDeselectSpline< 65535 THEN
	sDeselectSpline:= concat(concat('G',TO_STRING(nDeselectSpline)),' '); ELSE sDeselectSpline:=''; END_IF
IF nDeselectCornerRed >0 AND nDeselectCornerRed < 65535 THEN
	sDeselectCornerRed:= concat(concat('G',TO_STRING(nDeselectCornerRed)),' '); ELSE sDeselectCornerRed:=''; END_IF
//sGCodeOut := Concat(Concat(CONCAT('G',nPathPrep),' G'),nPlane);
sGCodeOut := Concat(Concat(Concat(Concat(Concat(Concat(Concat(Concat(sPathPrep,sPlane),sCutterComp),sDeselectDiamProg),sZeroOffset),sContMode),sMeasureMode),sDeselectSpline),sDeselectCornerRed);

//Timer
fbUpdate();

END_PROGRAM

// ---- Machine System/PRGs/Bogie/BogieSettings/BogieSettings.TcPOU
PROGRAM BogieSettings
VAR
	SaveButtonReq : BOOL;
	Saving : bool;		
END_VAR

//set var global via hmi and keep persistient persistient

	WX1Settings();
	WX2Settings();
	WX3Settings();
	WX4Settings();

END_PROGRAM

// ---- Machine System/PRGs/Bogie/BogieSettings/WX1Settings.TcPOU
PROGRAM WX1Settings
VAR
	WX1A_CP1_Send : HMI_Setting_GVL;
	WX1A_CP2_Send : HMI_Setting_GVL;
	WX1A_CP3_Send : HMI_Setting_GVL;
	
	WX1B_CP1_Send : HMI_Setting_GVL;
	WX1B_CP2_Send : HMI_Setting_GVL;
	WX1B_CP3_Send : HMI_Setting_GVL;
	WX1Saving 	: BOOL;
	WX1Save 	: BOOL;
	
END_VAR
VAR PERSISTENT
	WX1A_CP1_HMI : CPABS_CI;
	WX1A_CP2_HMI : CPABS_CI;
	WX1A_CP3_HMI : CPABS_CI;
	
	WX1B_CP1_HMI : CPABS_CI;
	WX1B_CP2_HMI : CPABS_CI;
	WX1B_CP3_HMI : CPABS_CI;
	
END_VAR

//saves hmi persistent input into the GVL on save
IF WX1Save THEN
	WX1Saving:=1;
	WX1Save:=0;
END_IF

IF WX1Saving THEN
	WX1A_CP1_Send(In:=WX1A_CP1_HMI, Out=>GVL_CP.WX1A_CP1_CIn);
	WX1A_CP2_Send(In:=WX1A_CP2_HMI, Out=>GVL_CP.WX1A_CP2_CIn);
	WX1A_CP3_Send(IN:=WX1A_CP3_HMI, (*Out=>GVL_CP.WX1A_CP3_CI*));
	
	WX1B_CP1_Send(IN:=WX1B_CP1_HMI, Out=>GVL_CP.WX1B_CP1_CIn);
	WX1B_CP2_Send(In:=WX1B_CP2_HMI, Out=>GVL_CP.WX1B_CP2_CI);
	WX1B_CP3_Send(IN:=WX1B_CP3_HMI, (*Out=>GVL_CP.WX1B_CP3_CI*));
	WX1Saving :=0;
END_IF

END_PROGRAM

// ---- Machine System/PRGs/Bogie/BogieSettings/HMI_Setting_GVL.TcPOU
FUNCTION_BLOCK HMI_Setting_GVL
VAR_INPUT
	In : CPABS_CI;
	Save : BOOL;
END_VAR
VAR_OUTPUT
	Out : CpABS_CI;
	Saving : bool;
END_VAR
VAR
	
END_VAR

//WX1A_CP1
IF Save THEN
	Saving:=1;
	Save:=0;
END_IF
IF Saving THEN
	Out.MotorName			:= In.MotorName;
	OUt.ABSEncoderScaler_CI := In.ABSEncoderScaler_CI;
	Out.ABSEncoderZero_CI 	:= In.ABSEncoderZero_CI;
	Out.cntPulseSet_CI 		:= In.cntPulseSet_CI;
	Out.DisPerFPulley_CI 	:= In.DisPerFPulley_CI;
	Out.DisPerPulse_CI 		:= IN.DisPerPulse_CI;
	OUt.DistPerMRev_CI 		:= In.DistPerMRev_CI;
	Out.GearRatio_CI 		:= In.GearRatio_CI;
	Out.HomingSet_CI 		:= In.HomingSet_CI;
	Out.InputFilter_CI 		:= IN.InputFilter_CI;
	Out.Lead_CI 			:= In.Lead_CI;
	Out.Limit_NC_NO_CI 		:= In.Limit_NC_NO_CI;
	OUt.MechDriveType_CI 	:= In.MechDriveType_CI;
	Out.MoveABSTol_CI 		:= IN.MoveABSTol_CI;
	Out.PPRset_CI 			:= In.PPRset_CI;
	Out.SWLimit_Hi_CI 		:= In.SWLimit_Hi_CI;
	Out.SWLimit_Lo_CI 		:= In.SWLimit_Lo_CI;
	
	Saving:=0;
END_IF

END_FUNCTION_BLOCK

// ---- Machine System/PRGs/Bogie/BogieSettings/WX2Settings.TcPOU
PROGRAM WX2Settings
VAR
	WX2A_CP1_Send : HMI_Setting_GVL;
	WX2A_CP2_Send : HMI_Setting_GVL;
	WX2A_CP3_Send : HMI_Setting_GVL;
	
	WX2B_CP1_Send : HMI_Setting_GVL;
	WX2B_CP2_Send : HMI_Setting_GVL;
	WX2B_CP3_Send : HMI_Setting_GVL;
	WX2Save : BOOL;
	WX2Saving : BOOL;
END_VAR
VAR PERSISTENT
	WX2A_CP1_HMI : CPABS_CI;
	WX2A_CP2_HMI : CPABS_CI;
	WX2A_CP3_HMI : CPABS_CI;
	
	WX2B_CP1_HMI : CPABS_CI;
	WX2B_CP2_HMI : CPABS_CI;
	WX2B_CP3_HMI : CPABS_CI;
	
END_VAR

//saves hmi persistient input into the GVL on save
IF WX2Save THEN
	WX2Saving:=1;
	WX2Save :=0;
END_IF

IF WX2Saving THEN
	WX2A_CP1_Send(In:=WX2A_CP1_HMI, Out=>GVL_CP.WX2A_CP1_CI);
	WX2A_CP2_Send(In:=WX2A_CP2_HMI, Out=>GVL_CP.WX2A_CP2_CI);
	WX2A_CP3_Send(IN:=WX2A_CP3_HMI, Out=>GVL_CP.WX2A_CP3_CI);
	
	WX2B_CP1_Send(IN:=WX2B_CP1_HMI, Out=>GVL_CP.WX2B_CP1_CIn);
	WX2B_CP2_Send(In:=WX2B_CP2_HMI, Out=>GVL_CP.WX2B_CP2_CI);
	WX2B_CP3_Send(IN:=WX2B_CP3_HMI, Out=>GVL_CP.WX2B_CP3_CI);
	WX2saving:=0;
END_IF

END_PROGRAM

// ---- Machine System/PRGs/Bogie/BogieSettings/WX3Settings.TcPOU
PROGRAM WX3Settings
VAR
	WX3A_CP1_Send : HMI_Setting_GVL;
	WX3A_CP2_Send : HMI_Setting_GVL;
	WX3A_CP3_Send : HMI_Setting_GVL;
	
	WX3B_CP1_Send : HMI_Setting_GVL;
	WX3B_CP2_Send : HMI_Setting_GVL;
	WX3B_CP3_Send : HMI_Setting_GVL;
	WX3Saving 	: BOOL;
	WX3Save 	: BOOL;
	
END_VAR
VAR PERSISTENT
	WX3A_CP1_HMI : CPABS_CI;
	WX3A_CP2_HMI : CPABS_CI;
	WX3A_CP3_HMI : CPABS_CI;
	
	WX3B_CP1_HMI : CPABS_CI;
	WX3B_CP2_HMI : CPABS_CI;
	WX3B_CP3_HMI : CPABS_CI;
	
END_VAR

//saves hmi persistent input into the GVL on save
IF WX3Save THEN
	WX3Saving:=1;
	WX3Save:=0;
END_IF

IF WX3Saving THEN
	WX3A_CP1_Send(In:=WX3A_CP1_HMI, Out=>GVL_CP.WX3A_CP1_CI);
	WX3A_CP2_Send(In:=WX3A_CP2_HMI, Out=>GVL_CP.WX3A_Cp2_CI);
	WX3A_CP3_Send(IN:=WX3A_CP3_HMI, (*Out=>GVL_CP.WX3A_CP3_CI*));
	
	WX3B_CP1_Send(IN:=WX3B_CP1_HMI, Out=>GVL_CP.WX3B_CP1_CI);
	WX3B_CP2_Send(In:=WX3B_CP2_HMI, Out=>GVL_CP.WX3B_CP2_CI);
	WX3B_CP3_Send(IN:=WX3B_CP3_HMI, (*Out=>GVL_CP.WX3B_CP3_CI*));
	WX3Saving :=0;
END_IF

END_PROGRAM

// ---- Machine System/PRGs/Bogie/BogieSettings/WX4Settings.TcPOU
PROGRAM WX4Settings
VAR
	WX4A_CP1_Send : HMI_Setting_GVL;
	WX4A_CP2_Send : HMI_Setting_GVL;
	WX4A_CP3_Send : HMI_Setting_GVL;
	
	WX4B_CP1_Send : HMI_Setting_GVL;
	WX4B_CP2_Send : HMI_Setting_GVL;
	WX4B_CP3_Send : HMI_Setting_GVL;
	WX4Save : BOOL;
	WX4Saving :BOOL;
END_VAR
VAR PERSISTENT
	WX4A_CP1_HMI : CPABS_CI;
	WX4A_CP2_HMI : CPABS_CI;
	WX4A_CP3_HMI : CPABS_CI;
	
	WX4B_CP1_HMI : CPABS_CI;
	WX4B_CP2_HMI : CPABS_CI;
	WX4B_CP3_HMI : CPABS_CI;
	
END_VAR

//saves hmi persistent input into the GVL on save
IF WX4Save THEN
	WX4Saving:=1;
	WX4Save :=0;
END_IF

IF WX4Saving THEN
	WX4A_CP1_Send(In:=WX4A_CP1_HMI, Out=>GVL_CP.WX4A_CP1_CI);
	WX4A_CP2_Send(In:=WX4A_CP2_HMI, Out=>GVL_CP.WX4A_Cp2_CI);
	WX4A_CP3_Send(IN:=WX4A_CP3_HMI, (*=>GVL_CP.WX4A_CP3_CI*));
	
	WX4B_CP1_Send(IN:=WX4B_CP1_HMI, Out=>GVL_CP.WX4B_CP1_CI);
	WX4B_CP2_Send(In:=WX4B_CP2_HMI, Out=>GVL_CP.WX4B_CP2_CI);
	WX4B_CP3_Send(IN:=WX4B_CP3_HMI, (*Out=>GVL_CP.WX4B_CP3_CI*));
	WX4Saving:=0;
END_IF

END_PROGRAM

// ---- Machine System/PRGs/RollerDoors.TcPOU
PROGRAM RollerDoors
VAR
	FQ1_FB : FB_RollerDoor;
	FQ2_FB : FB_RollerDoor;
	FQ3_FB : FB_RollerDoor;
END_VAR

//The Bogies control FQ2 and FQ3 on SD1 and SD2, respectively. 
//the conveyors are controlling all other doors

//FQ1 shuttle Roller Door
IF GVL_Doors.FQ1.StatusOpenedInput THEN 
	GVL_Doors.FQ1.AutoOpenRequest := 0;
END_IF

IF GVL_Doors.FQ1.StatusClosedInput THEN 
	GVL_Doors.FQ1.AutoCloseRequest := 0;
END_IF

FQ1_FB(	AutoMode				:= GVL_HMI.AutoMode,
		ManualMode 				:= GVL_HMI.ManualMode,
		ManualDoorOpenRequest	:= GVL_Doors.FQ1.ManualOpenRequest,
		ManualDoorCloseRequest 	:= GVL_Doors.FQ1.ManualCloseRequest,
		AutoDoorOpenRequest 	:= GVL_Doors.FQ1.AutoOpenRequest,
		AutoDoorCloseRequest 	:= GVL_Doors.FQ1.AutoCloseRequest,);
		
GVL_Doors.FQ1.CommandOpenOutput		:= FQ1_FB.DoorOpenCommand;
GVL_Doors.FQ1.CommandCloseOutput	:= FQ1_FB.DoorCloseCommand;


//FQ2 SD1 Roller Door
IF GVL_Doors.FQ2.StatusOpenedInput THEN 
	GVL_Doors.FQ2.AutoOpenRequest := 0;
END_IF

IF GVL_Doors.FQ2.StatusClosedInput THEN 
	GVL_Doors.FQ2.AutoCloseRequest := 0;
END_IF

FQ2_FB(	AutoMode				:= GVL_HMI.AutoMode,
		ManualMode 				:= GVL_HMI.ManualMode,
		ManualDoorOpenRequest	:= GVL_Doors.FQ2.ManualOpenRequest,
		ManualDoorCloseRequest 	:= GVL_Doors.FQ2.ManualCloseRequest,
		AutoDoorOpenRequest 	:= GVL_Doors.FQ2.AutoOpenRequest,
		AutoDoorCloseRequest 	:= GVL_Doors.FQ2.AutoCloseRequest,);
		
GVL_Doors.FQ2.CommandOpenOutput		:= FQ2_FB.DoorOpenCommand;
GVL_Doors.FQ2.CommandCloseOutput	:= FQ2_FB.DoorCloseCommand;

//FQ3 SD2 Roller Door
IF GVL_Doors.FQ3.StatusOpenedInput THEN 
	GVL_Doors.FQ3.AutoOpenRequest := 0;
END_IF

IF GVL_Doors.FQ3.StatusClosedInput THEN 
	GVL_Doors.FQ3.AutoCloseRequest := 0;
END_IF
		
FQ3_FB(	AutoMode				:= GVL_HMI.AutoMode,
		ManualMode 				:= GVL_HMI.ManualMode,
		ManualDoorOpenRequest	:= GVL_Doors.FQ3.ManualOpenRequest,
		ManualDoorCloseRequest 	:= GVL_Doors.FQ3.ManualCloseRequest,
		AutoDoorOpenRequest 	:= GVL_Doors.FQ3.AutoOpenRequest,
		AutoDoorCloseRequest 	:= GVL_Doors.FQ3.AutoCloseRequest,);

GVL_Doors.FQ3.CommandOpenOutput		:= FQ3_FB.DoorOpenCommand;
GVL_Doors.FQ3.CommandCloseOutput	:= FQ3_FB.DoorCloseCommand;

END_PROGRAM

// ---- Machine System/FBs/FB_RollerDoor.TcPOU
FUNCTION_BLOCK FB_RollerDoor
VAR_INPUT
	AutoMode : BOOL;
	ManualMode : BOOL;
	ManualDoorOpenRequest : BOOL;
	ManualDoorCloseRequest : BOOL;
	AutoDoorOpenRequest : BOOL;
	AutoDoorCloseRequest : BOOL;
	test:bool;
END_VAR
VAR_OUTPUT
	DoorOpenCommand : BOOL;
	DoorCloseCommand : BOOL;
END_VAR
VAR
	ManualDoorOpenRequestRTRIG : R_TRIG;
	ManualDoorCloseRequestRTRIG : R_TRIG;
	AutoDoorOpenRequestRTRIG : R_TRIG;
	AutoDoorCloseRequestRTRIG : R_TRIG;
END_VAR

IF AutoMode THEN
	
	AutoDoorOpenRequestRTRIG(CLK := AutoDoorOpenRequest);
	AutoDoorCloseRequestRTRIG(CLK := AutoDoorCloseRequest);
	
	IF AutoDoorOpenRequestRTRIG.Q THEN
		DoorOpenCommand := 1;
		DoorCloseCommand := 0;
	ELSIF AutoDoorCloseRequestRTRIG.Q THEN
		DoorCloseCommand := 1;
		DoorOpenCommand := 0;
	END_IF
END_IF

IF ManualMode THEN
	
	ManualDoorOpenRequestRTRIG(CLK := ManualDoorOpenRequest);
	ManualDoorCloseRequestRTRIG(CLK := ManualDoorCloseRequest);
	
	IF ManualDoorOpenRequestRTRIG.Q THEN
		DoorOpenCommand := 1;
		DoorCloseCommand := 0;
	ELSIF ManualDoorCloseRequestRTRIG.Q THEN
		DoorCloseCommand := 1;
		DoorOpenCommand := 0;
	END_IF
END_IF

END_FUNCTION_BLOCK

// ---- Machine System/PRGs/PersonnelDoor.TcPOU
PROGRAM PersonnelDoor
VAR
	
END_VAR

IF GVL_Doors.QQ1.OpenButtonRequestInput THEN
	GVL_Doors.QQ1.AccessAreaRequest := 1;
	GVL_Doors.QQ1.OpenButtonLED_Output := 1;
	GVL_Doors.QQ1.OkToUnlockDoor := 1; //Remove this once ventalation is hooked up. Ventalation and styrene sensor level will determine when this gets turned on.
	ELSE
	GVL_Doors.QQ1.OpenButtonLED_Output := 0;
END_IF

GVL_Doors.QQ1.OkToUnlockDoorRTRIG(CLK := GVL_Doors.QQ1.OkToUnlockDoor);


IF GVL_Doors.QQ1.OkToUnlockDoorRTRIG.Q THEN
	GVL_Doors.QQ1.AccessAreaRequest := 0;
	GVL_Doors.QQ1.OpenButtonLED_Output := 0;
	GVL_Doors.QQ1.LockButtonLED_Output := 1;
	GVL_Doors.QQ1.LockOutput := 1;
END_IF

IF GVL_Doors.QQ1.LockButtonRequestInput THEN
	GVL_Doors.QQ1.LockOutput := 0;	
	GVL_Doors.QQ1.LockButtonLED_Output := 0;
	GVL_Doors.QQ1.OkToUnlockDoor := 0; //Remove this once ventalation is hooked up.
END_IF

END_PROGRAM

// ---- Machine System/PRGs/Heraus_Heater_Control.TcPOU
PROGRAM Heraus_Heater_Control

VAR_INPUT
		HMI_RECIPE_NUM : INT; // SELECTED RECIPE VALUE FROM HMI NUMERIC INPUT
		
		HERAUS_STATUS  : INT; // BINARY STATUS INFORMATION FROM HEATER CABINET.
							  // 0 = OFF
							  // 1 = SYSTEM STARTING
							  // 2 = POST HEATING GAS ON
							  // 3 = RUNNING
							  // 4 = STANDBY
END_VAR

VAR
	HERAUS_ESTOP_OK      AT %I*: BOOL; // ESTOP OK INTERLOCK RELAY STATE
	HERAUS_STATUS_B1     AT %I*: BOOL; // HEARAUS HEATER STATUS BIT 1
	HERAUS_STATUS_B2     AT %I*: BOOL; // HEARAUS HEATER STATUS BIT 2
	HERAUS_STATUS_B3     AT %I*: BOOL; // HEARAUS HEATER STATUS BIT 3
	RECIPE_VALUE_BIT_0   AT %Q*: BOOL; // BINARY VALUE 1 RECIPE SELECTION
	RECIPE_VALUE_BIT_1   AT %Q*: BOOL; // BINARY VALUE 2 RECIPE SELECTION
	RECIPE_VALUE_BIT_2   AT %Q*: BOOL; // BINARY VALUE 4 RECIPE SELECTION
	RECIPE_VALUE_BIT_3   AT %Q*: BOOL; // BINARY VALUE 8 RECIPE SELECTION
	RECIPE_VALUE_BIT_4   AT %Q*: BOOL; // BINARY VALUE 16 RECIPE SELECTION
		
END_VAR

// INITIALIZE HEATER STATUS TO 0
		HERAUS_STATUS := 0;
IF HERAUS_STATUS_B1 AND NOT HERAUS_STATUS_B2 AND NOT HERAUS_STATUS_B3 THEN
		HERAUS_STATUS := 1;
ELSIF HERAUS_STATUS_B2 AND NOT HERAUS_STATUS_B1 AND NOT HERAUS_STATUS_B3 THEN
		HERAUS_STATUS := 2;
ELSIF HERAUS_STATUS_B3 AND NOT HERAUS_STATUS_B1 AND NOT HERAUS_STATUS_B2 THEN
		HERAUS_STATUS := 3;
ELSIF HERAUS_STATUS_B3 AND HERAUS_STATUS_B1 AND NOT HERAUS_STATUS_B2 THEN
		HERAUS_STATUS := 4;
END_IF

CASE HMI_RECIPE_NUM OF 
     1 : RECIPE_VALUE_BIT_0 := TRUE; 
         RECIPE_VALUE_BIT_1 := FALSE; 
		 RECIPE_VALUE_BIT_2 := FALSE;
		 RECIPE_VALUE_BIT_3 := FALSE;
		 RECIPE_VALUE_BIT_4 := FALSE; 

     2 : RECIPE_VALUE_BIT_0 := FALSE; 
         RECIPE_VALUE_BIT_1 := TRUE;
		 RECIPE_VALUE_BIT_2 := FALSE;
		 RECIPE_VALUE_BIT_3 := FALSE;
		 RECIPE_VALUE_BIT_4 := FALSE; 

	 3 : RECIPE_VALUE_BIT_0 := TRUE; 
         RECIPE_VALUE_BIT_1 := TRUE;
		 RECIPE_VALUE_BIT_2 := FALSE;
		 RECIPE_VALUE_BIT_3 := FALSE;
		 RECIPE_VALUE_BIT_4 := FALSE; 
		 
	 4 : RECIPE_VALUE_BIT_0 := FALSE; 
         RECIPE_VALUE_BIT_1 := FALSE;
		 RECIPE_VALUE_BIT_2 := TRUE;
		 RECIPE_VALUE_BIT_3 := FALSE;
		 RECIPE_VALUE_BIT_4 := FALSE; 
		 
	 5 : RECIPE_VALUE_BIT_0 := TRUE; 
         RECIPE_VALUE_BIT_1 := FALSE;
		 RECIPE_VALUE_BIT_2 := TRUE;
		 RECIPE_VALUE_BIT_3 := FALSE;
		 RECIPE_VALUE_BIT_4 := FALSE; 

     6 : RECIPE_VALUE_BIT_0 := FALSE; 
         RECIPE_VALUE_BIT_1 := TRUE;
		 RECIPE_VALUE_BIT_2 := TRUE;
		 RECIPE_VALUE_BIT_3 := FALSE;
		 RECIPE_VALUE_BIT_4 := FALSE; 

	 7 : RECIPE_VALUE_BIT_0 := TRUE; 
         RECIPE_VALUE_BIT_1 := TRUE;
		 RECIPE_VALUE_BIT_2 := TRUE;
		 RECIPE_VALUE_BIT_3 := FALSE;
		 RECIPE_VALUE_BIT_4 := FALSE; 
		 
	 8 : RECIPE_VALUE_BIT_0 := FALSE; 
         RECIPE_VALUE_BIT_1 := FALSE;
		 RECIPE_VALUE_BIT_2 := FALSE;
		 RECIPE_VALUE_BIT_3 := TRUE;
		 RECIPE_VALUE_BIT_4 := FALSE; 
		 
	 9 : RECIPE_VALUE_BIT_0 := TRUE; 
         RECIPE_VALUE_BIT_1 := FALSE;
		 RECIPE_VALUE_BIT_2 := FALSE;
		 RECIPE_VALUE_BIT_3 := TRUE;
		 RECIPE_VALUE_BIT_4 := FALSE; 
		 
	10 : RECIPE_VALUE_BIT_0 := FALSE; 
         RECIPE_VALUE_BIT_1 := TRUE;
		 RECIPE_VALUE_BIT_2 := FALSE;
		 RECIPE_VALUE_BIT_3 := TRUE;
		 RECIPE_VALUE_BIT_4 := FALSE; 
		
ELSE 
	     RECIPE_VALUE_BIT_0 := FALSE; 
         RECIPE_VALUE_BIT_1 := FALSE;
		 RECIPE_VALUE_BIT_2 := FALSE;
		 RECIPE_VALUE_BIT_3 := FALSE;
		 RECIPE_VALUE_BIT_4 := FALSE; 
END_CASE;

END_PROGRAM

// ---- Machine System/PRGs/Conveyors/Input_Buffering.TcPOU
PROGRAM Input_Buffering
VAR
END_VAR

// DE-BOUNCE TIMER FOR GL1 LOW LIMIT SWITCH ON
GVL_CONVEYORS.GL1.Low_Limit_TimerOn (IN := GVL_CONVEYORS.GL1.Low_limit, PT := GVL_HMI.GL1LowLimitOnPresetTime);
GVL_CONVEYORS.GL1.Low_Limit_TimerOn_Done_Bit := GVL_CONVEYORS.GL1.Low_Limit_TimerOn.Q;
GVL_CONVEYORS.GL1.LOW_LIMIT_TIMER_ON_ELAPSED := GVL_CONVEYORS.GL1.Low_Limit_TimerOn.ET;
GVL_CONVEYORS.GL1.LIMIT_LOW_ON := GVL_CONVEYORS.GL1.Low_Limit_TimerOn_Done_Bit;

// DE-BOUNCE TIMER FOR GL1 HIGH LIMIT SWITCH ON
GVL_CONVEYORS.GL1.HIGH_Limit_TimerOn (IN := GVL_CONVEYORS.GL1.HIGH_Limit, PT := GVL_HMI. GL1LowLimitOffPresetTime);
GVL_CONVEYORS.GL1.HIGH_Limit_TimerOn_Done_Bit := GVL_CONVEYORS.GL1.HIGH_Limit_TimerOn.Q;
GVL_CONVEYORS.GL1.HIGH_LIMIT_TIMER_ON_ELAPSED := GVL_CONVEYORS.GL1.HIGH_Limit_TimerOn.ET;
GVL_CONVEYORS.GL1.LIMIT_HIGH_ON := GVL_CONVEYORS.GL1.HIGH_Limit_TimerOn_Done_Bit;

// DE-BOUNCE TIMER FOR GL1 LOW LIMIT SWITCH Off
GVL_CONVEYORS.GL1.Low_Limit_TimerOff (IN := NOT GVL_CONVEYORS.GL1.Low_limit, PT := GVL_HMI.GL1HighLimitOnPresetTime);
GVL_CONVEYORS.GL1.Low_Limit_TimerOff_Done_Bit := GVL_CONVEYORS.GL1.Low_Limit_TimerOff.Q;
GVL_CONVEYORS.GL1.LOW_LIMIT_TIMER_Off_ELAPSED := GVL_CONVEYORS.GL1.Low_Limit_TimerOff.ET;
GVL_CONVEYORS.GL1.LIMIT_LOW_Off := GVL_CONVEYORS.GL1.LOW_Limit_TimerOff_Done_Bit;

// DE-BOUNCE TIMER FOR GL1 HIGH LIMIT SWITCH Off
GVL_CONVEYORS.GL1.HIGH_Limit_TimerOff (IN := NOT GVL_CONVEYORS.GL1.High_Limit, PT := GVL_HMI.GL1HighLimitOffPresetTime );
GVL_CONVEYORS.GL1.HIGH_Limit_TimerOff_Done_Bit := GVL_CONVEYORS.GL1.HIGH_Limit_TimerOff.Q;
GVL_CONVEYORS.GL1.HIGH_LIMIT_TIMER_Off_ELAPSED := GVL_CONVEYORS.GL1.HIGH_Limit_TimerOff.ET;
GVL_CONVEYORS.GL1.LIMIT_HIgh_OFF := GVL_CONVEYORS.GL1.HIGH_Limit_TimerOFF_Done_Bit;

// DE-BOUNCE TIMER FOR GL2 ENTER SWITCH ON
GVL_CONVEYORS.GL2.PP_ENTER_ON_TimerOn (IN := GVL_CONVEYORS.GL2.PP_Enter_left, PT := GVL_HMI.GL2PPEnterOnPresetTime);
GVL_CONVEYORS.GL2.PP_ENTER_ON_TimerOn_Done_Bit := GVL_CONVEYORS.GL2.PP_ENTER_ON_TimerOn.Q;
GVL_CONVEYORS.GL2.PP_ENTER_ON_TimerOn_ELAPSED := GVL_CONVEYORS.GL2.PP_ENTER_ON_TimerOn.ET;
GVL_CONVEYORS.GL2.Enter_Switch_is_on  := GVL_CONVEYORS.GL2.PP_ENTER_ON_TimerOn_Done_Bit;

// DE-BOUNCE TIMER FOR GL2 ENTER SWITCH OFF
GVL_CONVEYORS.GL2.PP_ENTER_OFF_TimerOff (IN := NOT GVL_CONVEYORS.GL2.PP_Enter_left, PT := GVL_HMI.GL2PPEnterOFFPresetTime);
GVL_CONVEYORS.GL2.PP_ENTER_OFF_TimerOff_Done_Bit := GVL_CONVEYORS.GL2.PP_ENTER_OFF_TimerOff.Q;
GVL_CONVEYORS.GL2.PP_ENTER_OFF_TimerOff_ELAPSED := GVL_CONVEYORS.GL2.PP_ENTER_OFF_TimerOff.ET;
GVL_CONVEYORS.GL2.Enter_Switch_is_Off  := GVL_CONVEYORS.GL2.PP_ENTER_OFF_TimerOff_Done_Bit;

// DE-BOUNCE TIMER FOR GL2 PP EXIT SWITCH ON
GVL_CONVEYORS.GL2.PP_EXIT_ON_TimerOn (IN := GVL_CONVEYORS.GL2.PP_EXIT_left, PT :=  GVL_HMI.GL2PPExitOnPresetTime);
GVL_CONVEYORS.GL2.PP_EXIT_ON_TimerOn_Done_Bit := GVL_CONVEYORS.GL2.PP_EXIT_ON_TimerOn.Q;
GVL_CONVEYORS.GL2.PP_EXIT_ON_TimerOn_ELAPSED := GVL_CONVEYORS.GL2.PP_EXIT_ON_TimerOn.ET;
GVL_CONVEYORS.GL2.EXIT_SWITCH_is_ON  := GVL_CONVEYORS.GL2.PP_EXIT_ON_TimerOn_Done_Bit;

// DE-BOUNCE TIMER FOR GL2 PP EXIT SWITCH OFF
GVL_CONVEYORS.GL2.PP_EXIT_OFF_TimerOff (IN :=  NOT GVL_CONVEYORS.GL2.PP_EXIT_left, PT := GVL_HMI.GL2PPExitOffPresetTime);
GVL_CONVEYORS.GL2.PP_EXIT_OFF_TimerOFF_Done_Bit := GVL_CONVEYORS.GL2.PP_EXIT_OFF_TimerOFF.Q;
GVL_CONVEYORS.GL2.PP_EXIT_OFF_TimerOFF_ELAPSED := GVL_CONVEYORS.GL2.PP_EXIT_OFF_TimerOFF.ET;
GVL_CONVEYORS.GL2.EXIT_SWITCH_is_OFF  := GVL_CONVEYORS.GL2.PP_EXIT_OFF_TimerOff_Done_Bit;

// DE-BOUNCE TIMER FOR GL2 AT GL5B PROX 1 POSITION SWITCH ON
GVL_CONVEYORS.GL2.AT_GL5B_PROX_1_ON_TimerOn (IN := GVL_CONVEYORS.GL2.At_GL5B_Prox_1, PT := GVL_HMI.GL2ATGl5BPositionProx1OnPresetTime);
GVL_CONVEYORS.GL2.AT_GL5B_PROX_1_ON_TimerOn_Done_Bit := GVL_CONVEYORS.GL2.AT_GL5B_PROX_1_ON_TimerOn.Q;
GVL_CONVEYORS.GL2.AT_GL5B_PROX_1_ON_TimerOn_ELAPSED := GVL_CONVEYORS.GL2.AT_GL5B_PROX_1_ON_TimerOn.ET;
GVL_CONVEYORS.GL2.AT_GL5B_PROX_1_ON := GVL_CONVEYORS.GL2.AT_GL5B_PROX_1_ON_TIMERON_Done_Bit;

// DE-BOUNCE TIMER FOR GL2 AT GL5B PROX 1 POSITION SWITCH OFF
GVL_CONVEYORS.GL2.AT_GL5B_PROX_1_OFF_TimerOff (IN := NOT GVL_CONVEYORS.GL2.At_GL5B_Prox_1, PT := GVL_HMI.GL2ATGl5BPositionProx1OffPresetTime);
GVL_CONVEYORS.GL2.AT_GL5B_PROX_1_OFF_TimerOff_Done_Bit := GVL_CONVEYORS.GL2.AT_GL5B_PROX_1_OFF_TimerOff.Q;
GVL_CONVEYORS.GL2.AT_GL5B_PROX_1_OFF_TimerOff_ELAPSED := GVL_CONVEYORS.GL2.AT_GL5B_PROX_1_OFF_TimerOff.ET;
GVL_CONVEYORS.GL2.AT_GL5B_PROX_1_OFF  := GVL_CONVEYORS.GL2.AT_GL5B_PROX_1_OFF_TimerOff_Done_Bit;

// DE-BOUNCE TIMER FOR GL2 AT GL5B PROX 2 POSITION SWITCH ON
GVL_CONVEYORS.GL2.AT_GL5B_PROX_2_ON_TimerOn (IN := GVL_CONVEYORS.GL2.At_GL5B_Prox_2, PT := GVL_HMI.GL2ATGl5BPositionProx2OnPresetTime);
GVL_CONVEYORS.GL2.AT_GL5B_PROX_2_ON_TimerOn_Done_Bit := GVL_CONVEYORS.GL2.AT_GL5B_PROX_2_ON_TimerOn.Q;
GVL_CONVEYORS.GL2.AT_GL5B_PROX_2_ON_TimerOn_ELAPSED := GVL_CONVEYORS.GL2.AT_GL5B_PROX_2_ON_TimerOn.ET;
GVL_CONVEYORS.GL2.AT_GL5B_PROX_2_ON := GVL_CONVEYORS.GL2.AT_GL5B_PROX_2_ON_TimerOn_Done_Bit;

// DE-BOUNCE TIMER FOR GL2 AT GL5B PROX 2 POSITION SWITCH OFF
GVL_CONVEYORS.GL2.AT_GL5B_PROX_2_OFF_TimerOff (IN := NOT GVL_CONVEYORS.GL2.AT_GL5B_PROX_2, PT := GVL_HMI.GL2ATGl5BPositionProx2OffPresetTime);
GVL_CONVEYORS.GL2.AT_GL5B_PROX_2_OFF_TimerOff_Done_Bit := GVL_CONVEYORS.GL2.AT_GL5B_PROX_2_OFF_TimerOff.Q;
GVL_CONVEYORS.GL2.AT_GL5B_PROX_2_OFF_TimerOff_ELAPSED := GVL_CONVEYORS.GL2.AT_GL5B_PROX_2_OFF_TimerOff.ET;
GVL_CONVEYORS.GL2.AT_GL5B_PROX_2_OFF := GVL_CONVEYORS.GL2.AT_GL5B_PROX_2_OFF_TimerOff_Done_Bit;

// DE-BOUNCE TIMER FOR GL2 AT GL6 PROX 1 POSITION SWITCH ON
GVL_CONVEYORS.GL2.AT_GL6_PROX_1_ON_TimerOn (IN := GVL_CONVEYORS.GL2.AT_GL6_PROX_1, PT := GVL_HMI.GL2ATGl6PositionProx1OnPresetTime);
GVL_CONVEYORS.GL2.AT_GL6_PROX_1_ON_TimerOn_Done_Bit := GVL_CONVEYORS.GL2.AT_GL6_PROX_1_ON_TimerON.Q;
GVL_CONVEYORS.GL2.AT_GL6_PROX_1_ON_TimerOn_ELAPSED := GVL_CONVEYORS.GL2.AT_GL6_PROX_1_ON_TimerOn.ET;
GVL_CONVEYORS.GL2.AT_GL6_PROX_1_ON := GVL_CONVEYORS.GL2.AT_GL6_PROX_1_ON_TimerOn_Done_Bit;

// DE-BOUNCE TIMER FOR GL2 AT GL6 PROX 1 POSITION SWITCH OFF
GVL_CONVEYORS.GL2.AT_GL6_PROX_1_OFF_TimerOff (IN := NOT GVL_CONVEYORS.GL2.AT_GL6_PROX_1, PT := GVL_HMI.GL2ATGl6PositionProx1OffPresetTime);
GVL_CONVEYORS.GL2.AT_GL6_PROX_1_OFF_TimerOff_Done_Bit := GVL_CONVEYORS.GL2.AT_GL6_PROX_1_OFF_TimerOff.Q;
GVL_CONVEYORS.GL2.AT_GL6_PROX_1_OFF_TimerOff_ELAPSED := GVL_CONVEYORS.GL2.AT_GL6_PROX_1_OFF_TimerOff.ET;
GVL_CONVEYORS.GL2.AT_GL6_PROX_1_OFF  := GVL_CONVEYORS.GL2.AT_GL6_PROX_1_OFF_TimerOff_Done_Bit;

// DE-BOUNCE TIMER FOR GL2 AT GL6 PROX 2 POSITION SWITCH ON
GVL_CONVEYORS.GL2.AT_GL6_PROX_2_ON_TimerOn (IN := GVL_CONVEYORS.GL2.AT_GL6_PROX_2, PT := GVL_HMI.GL2ATGl6PositionProx2OnPresetTime);
GVL_CONVEYORS.GL2.AT_GL6_PROX_2_ON_TimerOn_Done_Bit := GVL_CONVEYORS.GL2.AT_GL6_PROX_2_ON_TimerON.Q;
GVL_CONVEYORS.GL2.AT_GL6_PROX_2_ON_TimerOn_ELAPSED := GVL_CONVEYORS.GL2.AT_GL6_PROX_2_ON_TimerOn.ET;
GVL_CONVEYORS.GL2.AT_GL6_PROX_2_ON := GVL_CONVEYORS.GL2.AT_GL6_PROX_2_ON_TimerOn_Done_Bit;

// DE-BOUNCE TIMER FOR GL2 AT GL6 PROX 2 POSITION SWITCH OFF
GVL_CONVEYORS.GL2.AT_GL6_PROX_2_OFF_TimerOff (IN := NOT GVL_CONVEYORS.GL2.AT_GL6_PROX_2, PT := GVL_HMI.GL2ATGl6PositionProx2OffPresetTime);
GVL_CONVEYORS.GL2.AT_GL6_PROX_2_OFF_TimerOff_Done_Bit := GVL_CONVEYORS.GL2.AT_GL6_PROX_2_OFF_TimerOff.Q;
GVL_CONVEYORS.GL2.AT_GL6_PROX_2_OFF_TimerOff_ELAPSED := GVL_CONVEYORS.GL2.AT_GL6_PROX_2_OFF_TimerOff.ET;
GVL_CONVEYORS.GL2.AT_GL6_PROX_2_OFF  := GVL_CONVEYORS.GL2.AT_GL6_PROX_2_OFF_TimerOff_Done_Bit;

// DE-BOUNCE TIMER FOR GL2 AT GL8 PROX 1 POSITION SWITCH ON
GVL_CONVEYORS.GL2.AT_GL8_PROX_1_ON_TimerOn (IN := GVL_CONVEYORS.GL2.AT_GL8_PROX_1, PT := GVL_HMI.GL2ATGl8PositionProx1OnPresetTime);
GVL_CONVEYORS.GL2.AT_GL8_PROX_1_ON_TimerOn_Done_Bit := GVL_CONVEYORS.GL2.AT_GL8_PROX_1_ON_TimerON.Q;
GVL_CONVEYORS.GL2.AT_GL8_PROX_1_ON_TimerOn_ELAPSED := GVL_CONVEYORS.GL2.AT_GL8_PROX_1_ON_TimerOn.ET;
GVL_CONVEYORS.GL2.AT_GL8_PROX_1_ON := GVL_CONVEYORS.GL2.AT_GL8_PROX_1_ON_TimerOn_Done_Bit;

// DE-BOUNCE TIMER FOR GL2 AT GL8 PROX 1 POSITION SWITCH OFF
GVL_CONVEYORS.GL2.AT_GL8_PROX_1_OFF_TimerOff (IN := NOT GVL_CONVEYORS.GL2.AT_GL8_PROX_1, PT := GVL_HMI.GL2ATGl8PositionProx1OffPresetTime);
GVL_CONVEYORS.GL2.AT_GL8_PROX_1_OFF_TimerOff_Done_Bit := GVL_CONVEYORS.GL2.AT_GL8_PROX_1_OFF_TimerOff.Q;
GVL_CONVEYORS.GL2.AT_GL8_PROX_1_OFF_TimerOff_ELAPSED := GVL_CONVEYORS.GL2.AT_GL8_PROX_1_OFF_TimerOff.ET;
GVL_CONVEYORS.GL2.AT_GL8_PROX_1_OFF  := GVL_CONVEYORS.GL2.AT_GL8_PROX_1_OFF_TimerOff_Done_Bit;

// DE-BOUNCE TIMER FOR GL2 AT GL8 PROX 2 POSITION SWITCH ON
GVL_CONVEYORS.GL2.AT_GL8_PROX_2_ON_TimerOn (IN := GVL_CONVEYORS.GL2.AT_GL8_PROX_2, PT := GVL_HMI.GL2ATGl8PositionProx2OnPresetTime);
GVL_CONVEYORS.GL2.AT_GL8_PROX_2_ON_TimerOn_Done_Bit := GVL_CONVEYORS.GL2.AT_GL8_PROX_2_ON_TimerON.Q;
GVL_CONVEYORS.GL2.AT_GL8_PROX_2_ON_TimerOn_ELAPSED := GVL_CONVEYORS.GL2.AT_GL8_PROX_2_ON_TimerOn.ET;
GVL_CONVEYORS.GL2.AT_GL8_PROX_2_ON := GVL_CONVEYORS.GL2.AT_GL8_PROX_2_ON_TimerOn_Done_Bit;

// DE-BOUNCE TIMER FOR GL2 AT GL8 PROX 2 POSITION SWITCH OFF
GVL_CONVEYORS.GL2.AT_GL8_PROX_2_OFF_TimerOff (IN := NOT GVL_CONVEYORS.GL2.AT_GL8_PROX_2, PT := GVL_HMI.GL2ATGl8PositionProx2OffPresetTime);
GVL_CONVEYORS.GL2.AT_GL8_PROX_2_OFF_TimerOff_Done_Bit := GVL_CONVEYORS.GL2.AT_GL8_PROX_2_OFF_TimerOff.Q;
GVL_CONVEYORS.GL2.AT_GL8_PROX_2_OFF_TimerOff_ELAPSED := GVL_CONVEYORS.GL2.AT_GL8_PROX_2_OFF_TimerOff.ET;
GVL_CONVEYORS.GL2.AT_GL8_PROX_2_OFF  := GVL_CONVEYORS.GL2.AT_GL8_PROX_2_OFF_TimerOff_Done_Bit;

// DE-BOUNCE TIMER FOR GL3 PP ENTRY SWITCH ON
GVL_CONVEYORS.GL3.PP_ENTER_ON_TimerOn (IN := GVL_CONVEYORS.GL3.PP_ENTER_left, PT := GVL_HMI.GL3PPEnterOnPresetTime);
GVL_CONVEYORS.GL3.PP_ENTER_ON_TimerOn_Done_Bit := GVL_CONVEYORS.GL3.PP_ENTER_ON_TimerOn.Q;
GVL_CONVEYORS.GL3.PP_ENTER_ON_TimerOn_ELAPSED := GVL_CONVEYORS.GL3.PP_ENTER_ON_TimerOn.ET;
GVL_CONVEYORS.GL3.PP_ENTER_SWITCH_is_ON  := GVL_CONVEYORS.GL3.PP_ENTER_ON_TimerOn_Done_Bit;

// DE-BOUNCE TIMER FOR GL3 PP ENTRY SWITCH OFF
GVL_CONVEYORS.GL3.PP_ENTER_OFF_TimerOff (IN := NOT GVL_CONVEYORS.GL3.PP_Enter_left, PT := GVL_HMI.GL3PPEnterOffPresetTime);
GVL_CONVEYORS.GL3.PP_ENTER_OFF_TimerOFF_Done_Bit := GVL_CONVEYORS.GL3.PP_ENTER_OFF_TimerOFF.Q;
GVL_CONVEYORS.GL3.PP_ENTER_OFF_TimerOFF_ELAPSED := GVL_CONVEYORS.GL3.PP_ENTER_OFF_TimerOFF.ET;
GVL_CONVEYORS.GL3.PP_ENTER_SWITCH_is_OFF  := GVL_CONVEYORS.GL3.PP_ENTER_OFF_TimerOff_Done_Bit;

// DE-BOUNCE TIMER FOR GL3 PP EXIT SWITCH ON
GVL_CONVEYORS.GL3.PP_EXIT_ON_TimerOn (IN := GVL_CONVEYORS.GL3.PP_EXIT_LEFT, PT := GVL_HMI.GL3PPExitOnPresetTime);
GVL_CONVEYORS.GL3.PP_EXIT_ON_TimerOn_Done_Bit := GVL_CONVEYORS.GL3.PP_EXIT_ON_TimerOn.Q;
GVL_CONVEYORS.GL3.PP_EXIT_ON_TimerOn_ELAPSED := GVL_CONVEYORS.GL3.PP_EXIT_ON_TimerOn.ET;
GVL_CONVEYORS.GL3.PP_EXIT_SWITCH_is_ON  := GVL_CONVEYORS.GL3.PP_EXIT_ON_TimerOn_Done_Bit;

// DE-BOUNCE TIMER FOR GL3 PP EXIT SWITCH OFF
GVL_CONVEYORS.GL3.PP_EXIT_OFF_TimerOff (IN := NOT GVL_CONVEYORS.GL3.PP_EXIT_left, PT := GVL_HMI.GL3PPExitOffPresetTime);
GVL_CONVEYORS.GL3.PP_EXIT_OFF_TimerOFF_Done_Bit := GVL_CONVEYORS.GL3.PP_EXIT_OFF_TimerOFF.Q;
GVL_CONVEYORS.GL3.PP_EXIT_OFF_TimerOFF_ELAPSED := GVL_CONVEYORS.GL3.PP_EXIT_OFF_TimerOFF.ET;
GVL_CONVEYORS.GL3.PP_EXIT_SWITCH_is_OFF  := GVL_CONVEYORS.GL3.PP_EXIT_OFF_TimerOff_Done_Bit;

// DE-BOUNCE TIMER FOR GL4 PP ENTER SWITCH ON
GVL_CONVEYORS.GL4.PP_ENTER_ON_TimerOn (IN := GVL_CONVEYORS.GL4.PP_ENTER_left, PT := GVL_HMI.GL4PPEnterOnPresetTime);
GVL_CONVEYORS.GL4.PP_ENTER_ON_TimerOn_Done_Bit := GVL_CONVEYORS.GL4.PP_ENTER_ON_TimerOn.Q;
GVL_CONVEYORS.GL4.PP_ENTER_ON_TimerOn_ELAPSED := GVL_CONVEYORS.GL4.PP_ENTER_ON_TimerOn.ET;
GVL_CONVEYORS.GL4.PP_ENTER_SWITCH_is_ON  := GVL_CONVEYORS.GL4.PP_ENTER_ON_TimerOn_Done_Bit;

// DE-BOUNCE TIMER FOR GL4 PP ENTER SWITCH OFF
GVL_CONVEYORS.GL4.PP_ENTER_OFF_TimerOff (IN := NOT GVL_CONVEYORS.GL4.PP_Enter_left, PT :=GVL_HMI.GL4PPEnterOffPresetTime);
GVL_CONVEYORS.GL4.PP_ENTER_OFF_TimerOFF_Done_Bit := GVL_CONVEYORS.GL4.PP_ENTER_OFF_TimerOFF.Q;
GVL_CONVEYORS.GL4.PP_ENTER_OFF_TimerOFF_ELAPSED := GVL_CONVEYORS.GL4.PP_ENTER_OFF_TimerOFF.ET;
GVL_CONVEYORS.GL4.PP_ENTER_SWITCH_is_OFF  := GVL_CONVEYORS.GL4.PP_ENTER_OFF_TimerOff_Done_Bit;

// DE-BOUNCE TIMER FOR GL4 PP EXIT SWITCH ON
GVL_CONVEYORS.GL4.PP_EXIT_ON_TimerOn (IN := GVL_CONVEYORS.GL4.PP_EXIT_left, PT := GVL_HMI.GL4PPExitOnPresetTime);
GVL_CONVEYORS.GL4.PP_EXIT_ON_TimerOn_Done_Bit := GVL_CONVEYORS.GL4.PP_EXIT_ON_TimerOn.Q;
GVL_CONVEYORS.GL4.PP_EXIT_ON_TimerOn_ELAPSED := GVL_CONVEYORS.GL4.PP_EXIT_ON_TimerOn.ET;
GVL_CONVEYORS.GL4.PP_EXIT_SWITCH_is_ON  := GVL_CONVEYORS.GL4.PP_EXIT_ON_TimerOn_Done_Bit;

// DE-BOUNCE TIMER FOR GL4 PP EXIT SWITCH OFF
GVL_CONVEYORS.GL4.PP_EXIT_OFF_TimerOff (IN := NOT GVL_CONVEYORS.GL4.PP_EXIT_left, PT := GVL_HMI.GL4PPExitOffPresetTime);
GVL_CONVEYORS.GL4.PP_EXIT_OFF_TimerOFF_Done_Bit := GVL_CONVEYORS.GL4.PP_EXIT_OFF_TimerOFF.Q;
GVL_CONVEYORS.GL4.PP_EXIT_OFF_TimerOFF_ELAPSED := GVL_CONVEYORS.GL4.PP_EXIT_OFF_TimerOFF.ET;
GVL_CONVEYORS.GL4.PP_EXIT_SWITCH_is_OFF  := GVL_CONVEYORS.GL4.PP_EXIT_OFF_TimerOff_Done_Bit;

// DE-BOUNCE TIMER FOR GL5A PP ENTER SWITCH ON
GVL_CONVEYORS.GL5A.PP_ENTER_ON_TimerOn (IN := GVL_CONVEYORS.GL5A.PP_ENTER_left, PT := GVL_HMI.GL5APPEnterOnPresetTime);
GVL_CONVEYORS.GL5A.PP_ENTER_ON_TimerOn_Done_Bit := GVL_CONVEYORS.GL5A.PP_ENTER_ON_TimerOn.Q;
GVL_CONVEYORS.GL5A.PP_ENTER_ON_TimerOn_ELAPSED := GVL_CONVEYORS.GL5A.PP_ENTER_ON_TimerOn.ET;
GVL_CONVEYORS.GL5A.PP_ENTER_SWITCH_is_ON  := GVL_CONVEYORS.GL5A.PP_ENTER_ON_TimerOn_Done_Bit;

// DE-BOUNCE TIMER FOR GL5A PP ENTER SWITCH OFF
GVL_CONVEYORS.GL5A.PP_ENTER_OFF_TimerOff (IN := NOT GVL_CONVEYORS.GL5A.PP_Enter_left, PT := GVL_HMI.GL5APPEnterOffPresetTime);
GVL_CONVEYORS.GL5A.PP_ENTER_OFF_TimerOFF_Done_Bit := GVL_CONVEYORS.GL5A.PP_ENTER_OFF_TimerOFF.Q;
GVL_CONVEYORS.GL5A.PP_ENTER_OFF_TimerOFF_ELAPSED := GVL_CONVEYORS.GL5A.PP_ENTER_OFF_TimerOFF.ET;
GVL_CONVEYORS.GL5A.PP_ENTER_SWITCH_IS_OFF  := GVL_CONVEYORS.GL5A.PP_ENTER_OFF_TimerOff_Done_Bit;

// DE-BOUNCE TIMER FOR GL5A PP EXIT SWITCH ON
GVL_CONVEYORS.GL5A.PP_EXIT_ON_TimerOn (IN := GVL_CONVEYORS.GL5A.PP_EXIT_left, PT := GVL_HMI.GL5APPExitOnPresetTime);
GVL_CONVEYORS.GL5A.PP_EXIT_ON_TimerOn_Done_Bit := GVL_CONVEYORS.GL5A.PP_EXIT_ON_TimerOn.Q;
GVL_CONVEYORS.GL5A.PP_EXIT_ON_TimerOn_ELAPSED := GVL_CONVEYORS.GL5A.PP_EXIT_ON_TimerOn.ET;
GVL_CONVEYORS.GL5A.PP_Exit_Switch_Is_On  := GVL_CONVEYORS.GL5A.PP_EXIT_ON_TimerOn_Done_Bit;

// DE-BOUNCE TIMER FOR GL5A PP EXIT SWITCH OFF
GVL_CONVEYORS.GL5A.PP_EXIT_OFF_TimerOff (IN := NOT GVL_CONVEYORS.GL5A.PP_EXIT_left, PT := GVL_HMI.GL5APPExitOffPresetTime);
GVL_CONVEYORS.GL5A.PP_EXIT_OFF_TimerOFF_Done_Bit := GVL_CONVEYORS.GL5A.PP_EXIT_OFF_TimerOFF.Q;
GVL_CONVEYORS.GL5A.PP_EXIT_OFF_TimerOFF_ELAPSED := GVL_CONVEYORS.GL5A.PP_EXIT_OFF_TimerOFF.ET;
GVL_CONVEYORS.GL5A.PP_Exit_Switch_Is_Off  := GVL_CONVEYORS.GL5A.PP_EXIT_OFF_TimerOff_Done_Bit;

// DE-BOUNCE TIMER FOR GL5B PP ENTER SWITCH ON
GVL_CONVEYORS.GL5B.PP_ENTER_ON_TimerOn (IN := GVL_CONVEYORS.GL5B.PP_ENTER_left, PT := GVL_HMI.GL5BPPEnterOnPresetTime);
GVL_CONVEYORS.GL5B.PP_ENTER_ON_TimerOn_Done_Bit := GVL_CONVEYORS.GL5B.PP_ENTER_ON_TimerOn.Q;
GVL_CONVEYORS.GL5B.PP_ENTER_ON_TimerOn_ELAPSED := GVL_CONVEYORS.GL5B.PP_ENTER_ON_TimerOn.ET;
GVL_CONVEYORS.GL5B.PP_ENTER_SWITCH_is_ON  := GVL_CONVEYORS.GL5B.PP_ENTER_ON_TimerOn_Done_Bit;

// DE-BOUNCE TIMER FOR GL5B PP ENTER SWITCH OFF
GVL_CONVEYORS.GL5B.PP_ENTER_OFF_TimerOff (IN := NOT GVL_CONVEYORS.GL5B.PP_Enter_left, PT := GVL_HMI.GL5BPPEnterOffPresetTime);
GVL_CONVEYORS.GL5B.PP_ENTER_OFF_TimerOFF_Done_Bit := GVL_CONVEYORS.GL5B.PP_ENTER_OFF_TimerOFF.Q;
GVL_CONVEYORS.GL5B.PP_ENTER_OFF_TimerOFF_ELAPSED := GVL_CONVEYORS.GL5B.PP_ENTER_OFF_TimerOFF.ET;
GVL_CONVEYORS.GL5B.PP_ENTER_SWITCH_IS_OFF  := GVL_CONVEYORS.GL5B.PP_ENTER_OFF_TimerOff_Done_Bit;

// DE-BOUNCE TIMER FOR GL5B PP EXIT SWITCH ON
GVL_CONVEYORS.GL5B.PP_EXIT_ON_TimerOn (IN := GVL_CONVEYORS.GL5B.PP_EXIT_left, PT := GVL_HMI.GL5BPPExitOnPresetTime);
GVL_CONVEYORS.GL5B.PP_EXIT_ON_TimerOn_Done_Bit := GVL_CONVEYORS.GL5B.PP_EXIT_ON_TimerOn.Q;
GVL_CONVEYORS.GL5B.PP_EXIT_ON_TimerOn_ELAPSED := GVL_CONVEYORS.GL5B.PP_EXIT_ON_TimerOn.ET;
GVL_CONVEYORS.GL5B.PP_Exit_Switch_Is_On  := GVL_CONVEYORS.GL5B.PP_EXIT_ON_TimerOn_Done_Bit;

// DE-BOUNCE TIMER FOR GL5B PP EXIT SWITCH OFF
GVL_CONVEYORS.GL5B.PP_EXIT_OFF_TimerOff (IN := NOT GVL_CONVEYORS.GL5B.PP_EXIT_left, PT := GVL_HMI.GL5BPPExitOffPresetTime);
GVL_CONVEYORS.GL5B.PP_EXIT_OFF_TimerOFF_Done_Bit := GVL_CONVEYORS.GL5B.PP_EXIT_OFF_TimerOFF.Q;
GVL_CONVEYORS.GL5B.PP_EXIT_OFF_TimerOFF_ELAPSED := GVL_CONVEYORS.GL5B.PP_EXIT_OFF_TimerOFF.ET;
GVL_CONVEYORS.GL5B.PP_Exit_Switch_Is_Off  := GVL_CONVEYORS.GL5B.PP_EXIT_OFF_TimerOff_Done_Bit;

// DE-BOUNCE TIMER FOR GL6 PP ENTER SWITCH ON
GVL_CONVEYORS.GL6.PP_ENTER_ON_TimerOn (IN := GVL_CONVEYORS.GL6.PP_ENTER_left, PT := GVL_HMI.GL6PPEnterOnPresetTime);
GVL_CONVEYORS.GL6.PP_ENTER_ON_TimerOn_Done_Bit := GVL_CONVEYORS.GL6.PP_ENTER_ON_TimerOn.Q;
GVL_CONVEYORS.GL6.PP_ENTER_ON_TimerOn_ELAPSED := GVL_CONVEYORS.GL6.PP_ENTER_ON_TimerOn.ET;
GVL_CONVEYORS.GL6.PP_Enter_Switch_Is_On  := GVL_CONVEYORS.GL6.PP_ENTER_ON_TimerOn_Done_Bit;

// DE-BOUNCE TIMER FOR GL6 PP ENTER SWITCH OFF
GVL_CONVEYORS.GL6.PP_ENTER_OFF_TimerOff (IN := NOT GVL_CONVEYORS.GL6.PP_Enter_left, PT := GVL_HMI.GL6PPEnterOffPresetTime);
GVL_CONVEYORS.GL6.PP_ENTER_OFF_TimerOFF_Done_Bit := GVL_CONVEYORS.GL6.PP_ENTER_OFF_TimerOFF.Q;
GVL_CONVEYORS.GL6.PP_ENTER_OFF_TimerOFF_ELAPSED := GVL_CONVEYORS.GL6.PP_ENTER_OFF_TimerOFF.ET;
GVL_CONVEYORS.GL6.PP_ENTER_SWITCH_IS_OFF  := GVL_CONVEYORS.GL6.PP_ENTER_OFF_TimerOff_Done_Bit;

// DE-BOUNCE TIMER FOR GL6 PP EXIT SWITCH ON
GVL_CONVEYORS.GL6.PP_EXIT_ON_TimerOn (IN := GVL_CONVEYORS.GL6.PP_EXIT_left, PT := GVL_HMI.GL6PPExitOnPresetTime);
GVL_CONVEYORS.GL6.PP_EXIT_ON_TimerOn_Done_Bit := GVL_CONVEYORS.GL6.PP_EXIT_ON_TimerOn.Q;
GVL_CONVEYORS.GL6.PP_EXIT_ON_TimerOn_ELAPSED := GVL_CONVEYORS.GL6.PP_EXIT_ON_TimerOn.ET;
GVL_CONVEYORS.GL6.PP_EXIT_SWITCH_IS_ON  := GVL_CONVEYORS.GL6.PP_EXIT_ON_TimerOn_Done_Bit;

// DE-BOUNCE TIMER FOR GL6 PP EXIT SWITCH OFF
GVL_CONVEYORS.GL6.PP_EXIT_OFF_TimerOff (IN := NOT GVL_CONVEYORS.GL6.PP_EXIT_left, PT := GVL_HMI.GL6PPExitOffPresetTime);
GVL_CONVEYORS.GL6.PP_EXIT_OFF_TimerOFF_Done_Bit := GVL_CONVEYORS.GL6.PP_EXIT_OFF_TimerOFF.Q;
GVL_CONVEYORS.GL6.PP_EXIT_OFF_TimerOFF_ELAPSED := GVL_CONVEYORS.GL6.PP_EXIT_OFF_TimerOFF.ET;
GVL_CONVEYORS.GL6.PP_Exit_Switch_Is_Off  := GVL_CONVEYORS.GL6.PP_EXIT_OFF_TimerOff_Done_Bit;

// DE-BOUNCE TIMER FOR GL6 LOAD POSITION 1 SWITCH ON
GVL_CONVEYORS.GL6.LOAD_POS1_ON_TimerOn (IN := GVL_CONVEYORS.GL6.LOAD_POS_1, PT := GVL_HMI.GL6PPLoadPos1OnPresetTime);
GVL_CONVEYORS.GL6.LOAD_POS1_ON_TimerOn_Done_Bit := GVL_CONVEYORS.GL6.LOAD_POS1_ON_TimerOn.Q;
GVL_CONVEYORS.GL6.LOAD_POS1_ON_TimerOn_ELAPSED := GVL_CONVEYORS.GL6.LOAD_POS1_ON_TimerOn.ET;
GVL_CONVEYORS.GL6.PP_LOAD_POS_1_IS_ON  := GVL_CONVEYORS.GL6.LOAD_POS1_ON_TimerOn_Done_Bit;

// DE-BOUNCE TIMER FOR GL6 LOAD POSITION 1 SWITCH OFF
GVL_CONVEYORS.GL6.LOAD_POS1_OFF_TimerOff (IN := NOT GVL_CONVEYORS.GL6.LOAD_POS_1, PT := GVL_HMI.GL6PPLoadPos1OffPresetTime);
GVL_CONVEYORS.GL6.LOAD_POS1_OFF_TimerOFF_Done_Bit := GVL_CONVEYORS.GL6.LOAD_POS1_OFF_TimerOFF.Q;
GVL_CONVEYORS.GL6.LOAD_POS1_OFF_TimerOFF_ELAPSED := GVL_CONVEYORS.GL6.LOAD_POS1_OFF_TimerOFF.ET;
GVL_CONVEYORS.GL6.PP_LOAD_POS_1_IS_OFF  := GVL_CONVEYORS.GL6.LOAD_POS1_OFF_TimerOff_Done_Bit;

// DE-BOUNCE TIMER FOR GL6 LOAD POSITION 2 SWITCH ON
GVL_CONVEYORS.GL6.LOAD_POS2_ON_TimerOn (IN := GVL_CONVEYORS.GL6.LOAD_POS_2, PT := GVL_HMI.GL6PPLoadPos2OnPresetTime);
GVL_CONVEYORS.GL6.LOAD_POS2_ON_TimerOn_Done_Bit := GVL_CONVEYORS.GL6.LOAD_POS2_ON_TimerOn.Q;
GVL_CONVEYORS.GL6.LOAD_POS2_ON_TimerOn_ELAPSED := GVL_CONVEYORS.GL6.LOAD_POS2_ON_TimerOn.ET;
GVL_CONVEYORS.GL6.PP_LOAD_POS_2_IS_ON  := GVL_CONVEYORS.GL6.LOAD_POS2_ON_TimerOn_Done_Bit;

// DE-BOUNCE TIMER FOR GL6 LOAD POSITION 2 SWITCH OFF
GVL_CONVEYORS.GL6.LOAD_POS2_OFF_TimerOff (IN := NOT GVL_CONVEYORS.GL6.LOAD_POS_2, PT := GVL_HMI.GL6PPLoadPos2OffPresetTime);
GVL_CONVEYORS.GL6.LOAD_POS2_OFF_TimerOFF_Done_Bit := GVL_CONVEYORS.GL6.LOAD_POS2_OFF_TimerOFF.Q;
GVL_CONVEYORS.GL6.LOAD_POS2_OFF_TimerOFF_ELAPSED := GVL_CONVEYORS.GL6.LOAD_POS2_OFF_TimerOFF.ET;
GVL_CONVEYORS.GL6.PP_LOAD_POS_2_IS_OFF  := GVL_CONVEYORS.GL6.LOAD_POS2_OFF_TimerOff_Done_Bit;

// DE-BOUNCE TIMER FOR GL7 PP ENTER SWITCH ON
GVL_CONVEYORS.GL7.PP_ENTER_ON_TimerOn (IN := GVL_CONVEYORS.GL7.PP_ENTER_left, PT := GVL_HMI.GL7PPEnterOnPresetTime);
GVL_CONVEYORS.GL7.PP_ENTER_ON_TimerOn_Done_Bit := GVL_CONVEYORS.GL7.PP_ENTER_ON_TimerOn.Q;
GVL_CONVEYORS.GL7.PP_ENTER_ON_TimerOn_ELAPSED := GVL_CONVEYORS.GL7.PP_ENTER_ON_TimerOn.ET;
GVL_CONVEYORS.GL7.PP_ENTER_SWITCH_IS_ON  := GVL_CONVEYORS.GL7.PP_ENTER_ON_TimerOn_Done_Bit;

// DE-BOUNCE TIMER FOR GL7 PP ENTER SWITCH OFF
GVL_CONVEYORS.GL7.PP_ENTER_OFF_TimerOff (IN := NOT GVL_CONVEYORS.GL7.PP_Enter_left, PT := GVL_HMI.GL7PPEnterOffPresetTime);
GVL_CONVEYORS.GL7.PP_ENTER_OFF_TimerOFF_Done_Bit := GVL_CONVEYORS.GL7.PP_ENTER_OFF_TimerOFF.Q;
GVL_CONVEYORS.GL7.PP_ENTER_OFF_TimerOFF_ELAPSED := GVL_CONVEYORS.GL7.PP_ENTER_OFF_TimerOFF.ET;
GVL_CONVEYORS.GL7.PP_ENTER_SWITCH_IS_OFF  := GVL_CONVEYORS.GL7.PP_ENTER_OFF_TimerOff_Done_Bit;

// DE-BOUNCE TIMER FOR GL7 PP EXIT SWITCH ON
GVL_CONVEYORS.GL7.PP_EXIT_ON_TimerOn (IN := GVL_CONVEYORS.GL7.PP_EXIT_left, PT := GVL_HMI.GL7PPExitOnPresetTime);
GVL_CONVEYORS.GL7.PP_EXIT_ON_TimerOn_Done_Bit := GVL_CONVEYORS.GL7.PP_EXIT_ON_TimerOn.Q;
GVL_CONVEYORS.GL7.PP_EXIT_ON_TimerOn_ELAPSED := GVL_CONVEYORS.GL7.PP_EXIT_ON_TimerOn.ET;
GVL_CONVEYORS.GL7.PP_EXIT_SWITCH_IS_ON  := GVL_CONVEYORS.GL7.PP_EXIT_ON_TimerOn_Done_Bit;

// DE-BOUNCE TIMER FOR GL7 PP EXIT SWITCH OFF
GVL_CONVEYORS.GL7.PP_EXIT_OFF_TimerOff (IN := NOT GVL_CONVEYORS.GL7.PP_EXIT_left, PT := GVL_HMI.GL7PPExitOffPresetTime);
GVL_CONVEYORS.GL7.PP_EXIT_OFF_TimerOFF_Done_Bit := GVL_CONVEYORS.GL7.PP_EXIT_OFF_TimerOFF.Q;
GVL_CONVEYORS.GL7.PP_EXIT_OFF_TimerOFF_ELAPSED := GVL_CONVEYORS.GL7.PP_EXIT_OFF_TimerOFF.ET;
GVL_CONVEYORS.GL7.PP_EXIT_SWITCH_IS_OFF  := GVL_CONVEYORS.GL7.PP_EXIT_OFF_TimerOff_Done_Bit;

// DE-BOUNCE TIMER FOR GL8 PP ENTER SWITCH ON
GVL_CONVEYORS.GL8.PP_ENTER_ON_TimerOn (IN := GVL_CONVEYORS.GL8.PP_ENTER_RIGHT, PT := GVL_HMI.GL8PPEnterOnPresetTime);
GVL_CONVEYORS.GL8.PP_ENTER_ON_TimerOn_Done_Bit := GVL_CONVEYORS.GL8.PP_ENTER_ON_TimerOn.Q;
GVL_CONVEYORS.GL8.PP_ENTER_ON_TimerOn_ELAPSED := GVL_CONVEYORS.GL8.PP_ENTER_ON_TimerOn.ET;
GVL_CONVEYORS.GL8.PP_ENTER_SWITCH_IS_ON  := GVL_CONVEYORS.GL8.PP_ENTER_ON_TimerOn_Done_Bit;

// DE-BOUNCE TIMER FOR GL8 PP ENTER SWITCH OFF
GVL_CONVEYORS.GL8.PP_ENTER_OFF_TimerOff (IN := NOT GVL_CONVEYORS.GL8.PP_Enter_left, PT := GVL_HMI.GL8PPEnterOffPresetTime);
GVL_CONVEYORS.GL8.PP_ENTER_OFF_TimerOFF_Done_Bit := GVL_CONVEYORS.GL8.PP_ENTER_OFF_TimerOFF.Q;
GVL_CONVEYORS.GL8.PP_ENTER_OFF_TimerOFF_ELAPSED := GVL_CONVEYORS.GL8.PP_ENTER_OFF_TimerOFF.ET;
GVL_CONVEYORS.GL8.PP_ENTER_SWITCH_IS_OFF  := GVL_CONVEYORS.GL8.PP_ENTER_OFF_TimerOff_Done_Bit;

// DE-BOUNCE TIMER FOR GL8 PP EXIT SWITCH ON
GVL_CONVEYORS.GL8.PP_EXIT_ON_TimerOn (IN := GVL_CONVEYORS.GL8.PP_EXIT_left, PT := GVL_HMI.GL8PPExitOnPresetTime);
GVL_CONVEYORS.GL8.PP_EXIT_ON_TimerOn_Done_Bit := GVL_CONVEYORS.GL8.PP_EXIT_ON_TimerOn.Q;
GVL_CONVEYORS.GL8.PP_EXIT_ON_TimerOn_ELAPSED := GVL_CONVEYORS.GL8.PP_EXIT_ON_TimerOn.ET;
GVL_CONVEYORS.GL8.PP_EXIT_SWITCH_IS_ON  := GVL_CONVEYORS.GL8.PP_EXIT_ON_TimerOn_Done_Bit;

// DE-BOUNCE TIMER FOR GL8 PP EXIT SWITCH OFF
GVL_CONVEYORS.GL8.PP_EXIT_OFF_TimerOff (IN := NOT GVL_CONVEYORS.GL8.PP_EXIT_left, PT := GVL_HMI.GL8PPExitOffPresetTime);
GVL_CONVEYORS.GL8.PP_EXIT_OFF_TimerOFF_Done_Bit := GVL_CONVEYORS.GL8.PP_EXIT_OFF_TimerOFF.Q;
GVL_CONVEYORS.GL8.PP_EXIT_OFF_TimerOFF_ELAPSED := GVL_CONVEYORS.GL8.PP_EXIT_OFF_TimerOFF.ET;
GVL_CONVEYORS.GL8.PP_EXIT_SWITCH_IS_OFF  := GVL_CONVEYORS.GL8.PP_EXIT_OFF_TimerOff_Done_Bit;

// DE-BOUNCE TIMER FOR GL8 LOAD POSITION 1 SWITCH ON
GVL_CONVEYORS.GL8.LOAD_POS1_ON_TimerOn (IN := GVL_CONVEYORS.GL8.LOAD_POS_1, PT := GVL_HMI.GL8PPLoadPos1OnPresetTime);
GVL_CONVEYORS.GL8.LOAD_POS1_ON_TimerOn_Done_Bit := GVL_CONVEYORS.GL8.LOAD_POS1_ON_TimerOn.Q;
GVL_CONVEYORS.GL8.LOAD_POS1_ON_TimerOn_ELAPSED := GVL_CONVEYORS.GL8.LOAD_POS1_ON_TimerOn.ET;
GVL_CONVEYORS.GL8.PP_LOAD_POS_1_IS_ON  := GVL_CONVEYORS.GL8.LOAD_POS1_ON_TimerOn_Done_Bit;

// DE-BOUNCE TIMER FOR GL8 LOAD POSITION 1 SWITCH OFF
GVL_CONVEYORS.GL8.LOAD_POS1_OFF_TimerOff (IN := NOT GVL_CONVEYORS.GL8.LOAD_POS_1, PT := GVL_HMI.GL8PPLoadPos1OffPresetTime);
GVL_CONVEYORS.GL8.LOAD_POS1_OFF_TimerOFF_Done_Bit := GVL_CONVEYORS.GL8.LOAD_POS1_OFF_TimerOFF.Q;
GVL_CONVEYORS.GL8.LOAD_POS1_OFF_TimerOFF_ELAPSED := GVL_CONVEYORS.GL8.LOAD_POS1_OFF_TimerOFF.ET;
GVL_CONVEYORS.GL8.PP_LOAD_POS_1_IS_OFF  := GVL_CONVEYORS.GL8.LOAD_POS1_OFF_TimerOff_Done_Bit;

// DE-BOUNCE TIMER FOR GL8 LOAD POSITION 2 SWITCH ON
GVL_CONVEYORS.GL8.LOAD_POS2_ON_TimerOn (IN := GVL_CONVEYORS.GL8.LOAD_POS_2, PT := GVL_HMI.GL8PPLoadPos2OnPresetTime);
GVL_CONVEYORS.GL8.LOAD_POS2_ON_TimerOn_Done_Bit := GVL_CONVEYORS.GL8.LOAD_POS2_ON_TimerOn.Q;
GVL_CONVEYORS.GL8.LOAD_POS2_ON_TimerOn_ELAPSED := GVL_CONVEYORS.GL8.LOAD_POS2_ON_TimerOn.ET;
GVL_CONVEYORS.GL8.PP_LOAD_POS_2_IS_ON  := GVL_CONVEYORS.GL8.LOAD_POS2_ON_TimerOn_Done_Bit;

// DE-BOUNCE TIMER FOR GL8 LOAD POSITION 2 SWITCH OFF
GVL_CONVEYORS.GL8.LOAD_POS2_OFF_TimerOff (IN := NOT GVL_CONVEYORS.GL8.LOAD_POS_2, PT := GVL_HMI.GL8PPLoadPos2OffPresetTime);
GVL_CONVEYORS.GL8.LOAD_POS2_OFF_TimerOFF_Done_Bit := GVL_CONVEYORS.GL8.LOAD_POS2_OFF_TimerOFF.Q;
GVL_CONVEYORS.GL8.LOAD_POS2_OFF_TimerOFF_ELAPSED := GVL_CONVEYORS.GL8.LOAD_POS2_OFF_TimerOFF.ET;
GVL_CONVEYORS.GL8.PP_LOAD_POS_2_IS_OFF  := GVL_CONVEYORS.GL8.LOAD_POS2_OFF_TimerOff_Done_Bit;

// DE-BOUNCE TIMER FOR GL9 PP ENTER SWITCH ON
GVL_CONVEYORS.GL9.PP_ENTER_ON_TimerOn (IN := GVL_CONVEYORS.GL9.PP_ENTER_left, PT := GVL_HMI.GL9PPEnterOnPresetTime);
GVL_CONVEYORS.GL9.PP_ENTER_ON_TimerOn_Done_Bit := GVL_CONVEYORS.GL9.PP_ENTER_ON_TimerOn.Q;
GVL_CONVEYORS.GL9.PP_ENTER_ON_TimerOn_ELAPSED := GVL_CONVEYORS.GL9.PP_ENTER_ON_TimerOn.ET;
GVL_CONVEYORS.GL9.PP_ENTER_SWITCH_IS_ON  := GVL_CONVEYORS.GL9.PP_ENTER_ON_TimerOn_Done_Bit;

// DE-BOUNCE TIMER FOR GL9 PP ENTER SWITCH OFF
GVL_CONVEYORS.GL9.PP_ENTER_OFF_TimerOff (IN := NOT GVL_CONVEYORS.GL9.PP_Enter_left, PT := GVL_HMI.GL8PPEnterOffPresetTime);
GVL_CONVEYORS.GL9.PP_ENTER_OFF_TimerOFF_Done_Bit := GVL_CONVEYORS.GL9.PP_ENTER_OFF_TimerOFF.Q;
GVL_CONVEYORS.GL9.PP_ENTER_OFF_TimerOFF_ELAPSED := GVL_CONVEYORS.GL9.PP_ENTER_OFF_TimerOFF.ET;
GVL_CONVEYORS.GL9.PP_ENTER_SWITCH_IS_OFF  := GVL_CONVEYORS.GL9.PP_ENTER_OFF_TimerOff_Done_Bit;

// DE-BOUNCE TIMER FOR GL9 PP EXIT SWITCH ON
GVL_CONVEYORS.GL9.PP_EXIT_ON_TimerOn (IN := GVL_CONVEYORS.GL9.PP_EXIT_Left, PT := GVL_HMI.GL9PPExitOnPresetTime);
GVL_CONVEYORS.GL9.PP_EXIT_ON_TimerOn_Done_Bit := GVL_CONVEYORS.GL9.PP_EXIT_ON_TimerOn.Q;
GVL_CONVEYORS.GL9.PP_EXIT_ON_TimerOn_ELAPSED := GVL_CONVEYORS.GL9.PP_EXIT_ON_TimerOn.ET;
GVL_CONVEYORS.GL9.PP_EXIT_SWITCH_IS_ON  := GVL_CONVEYORS.GL9.PP_EXIT_ON_TimerOn_Done_Bit;

// DE-BOUNCE TIMER FOR GL9 PP EXIT SWITCH OFF
GVL_CONVEYORS.GL9.PP_EXIT_OFF_TimerOff (IN := NOT GVL_CONVEYORS.GL9.PP_EXIT_left, PT := GVL_HMI.GL9PPExitOffPresetTime);
GVL_CONVEYORS.GL9.PP_EXIT_OFF_TimerOFF_Done_Bit := GVL_CONVEYORS.GL9.PP_EXIT_OFF_TimerOFF.Q;
GVL_CONVEYORS.GL9.PP_EXIT_OFF_TimerOFF_ELAPSED := GVL_CONVEYORS.GL9.PP_EXIT_OFF_TimerOFF.ET;
GVL_CONVEYORS.GL9.PP_EXIT_SWITCH_IS_OFF  := GVL_CONVEYORS.GL9.PP_EXIT_OFF_TimerOff_Done_Bit;

// DE-BOUNCE TIMER FOR GL10 LOW LIMIT SWITCH ON
GVL_CONVEYORS.GL10.Low_Limit_TimerOn (IN := GVL_CONVEYORS.GL10.Low_Limit, PT := GVL_HMI.GL10LowLimitOnPresetTime);
GVL_CONVEYORS.GL10.Low_Limit_TimerOn_Done_Bit := GVL_CONVEYORS.GL10.Low_Limit_TimerOn.Q;
GVL_CONVEYORS.GL10.LOW_LIMIT_TIMER_ON_ELAPSED := GVL_CONVEYORS.GL10.Low_Limit_TimerOn.ET;
GVL_CONVEYORS.GL10.LIMIT_LOW_ON := GVL_CONVEYORS.GL10.Low_Limit_TimerOn_Done_Bit;

// DE-BOUNCE TIMER FOR GL10 LOW LIMIT SWITCH OFF
GVL_CONVEYORS.GL10.Low_Limit_TimerOff (IN := NOT GVL_CONVEYORS.GL10.LOW_limit, PT := GVL_HMI.GL10LowLimitOffPresetTime);
GVL_CONVEYORS.GL10.Low_Limit_TimerOff_Done_Bit := GVL_CONVEYORS.GL10.Low_Limit_TimerOff.Q;
GVL_CONVEYORS.GL10.LOW_LIMIT_TIMER_Off_ELAPSED := GVL_CONVEYORS.GL10.Low_Limit_TimerOff.ET;
GVL_CONVEYORS.GL10.LIMIT_LOW_OFF := GVL_CONVEYORS.GL10.LOW_Limit_TimerOFF_Done_Bit;

// DE-BOUNCE TIMER FOR GL10 HIGH LIMIT SWITCH ON
GVL_CONVEYORS.GL10.HIGH_Limit_TimerOn (IN := GVL_CONVEYORS.GL10.HIGH_limit, PT := GVL_HMI.GL10HighLimitOnPresetTime);
GVL_CONVEYORS.GL10.HIGH_Limit_TimerOn_Done_Bit := GVL_CONVEYORS.GL10.HIGH_Limit_TimerOn.Q;
GVL_CONVEYORS.GL10.HIGH_LIMIT_TIMER_ON_ELAPSED := GVL_CONVEYORS.GL10.HIGH_Limit_TimerOn.ET;
GVL_CONVEYORS.GL10.LIMIT_HIGH_ON := GVL_CONVEYORS.GL10.HIGH_Limit_TimerOn_Done_Bit;

// DE-BOUNCE TIMER FOR GL10 HIGH LIMIT SWITCH Off
GVL_CONVEYORS.GL10.HIGH_Limit_TimerOff (IN := NOT GVL_CONVEYORS.GL10.HIGH_LIMIT, PT := GVL_HMI.GL10HighLimitOffPresetTime);
GVL_CONVEYORS.GL10.HIGH_Limit_TimerOff_Done_Bit := GVL_CONVEYORS.GL10.HIGH_Limit_TimerOff.Q;
GVL_CONVEYORS.GL10.HIGH_LIMIT_TIMER_Off_ELAPSED := GVL_CONVEYORS.GL10.HIGH_Limit_TimerOff.ET;
GVL_CONVEYORS.GL10.LIMIT_HIGH_OFF := GVL_CONVEYORS.GL10.HIGH_Limit_TimerOFF_Done_Bit;


// DE-BOUNCE TIMER FOR GL11 PP ENTER SWITCH ON
GVL_CONVEYORS.GL11.PP_ENTER_ON_TimerOn (IN := GVL_CONVEYORS.GL11.PP_ENTER_left, PT := GVL_HMI.GL11PPEnterOnPresetTime);
GVL_CONVEYORS.GL11.PP_ENTER_ON_TimerOn_Done_Bit := GVL_CONVEYORS.GL11.PP_ENTER_ON_TimerOn.Q;
GVL_CONVEYORS.GL11.PP_ENTER_ON_TimerOn_ELAPSED := GVL_CONVEYORS.GL11.PP_ENTER_ON_TimerOn.ET;
GVL_CONVEYORS.GL11.ENTER_SWITCH_IS_ON  := GVL_CONVEYORS.GL11.PP_ENTER_ON_TimerOn_Done_Bit;

// DE-BOUNCE TIMER FOR GL11 PP ENTER SWITCH OFF
GVL_CONVEYORS.GL11.PP_ENTER_OFF_TimerOff (IN := NOT GVL_CONVEYORS.GL11.PP_ENTER_left, PT := GVL_HMI.GL11PPEnterOffPresetTime);
GVL_CONVEYORS.GL11.PP_ENTER_OFF_TimerOFF_Done_Bit := GVL_CONVEYORS.GL11.PP_ENTER_OFF_TimerOFF.Q;
GVL_CONVEYORS.GL11.PP_ENTER_OFF_TimerOFF_ELAPSED := GVL_CONVEYORS.GL11.PP_ENTER_OFF_TimerOFF.ET;
GVL_CONVEYORS.GL11.ENTER_SWITCH_IS_OFF  := GVL_CONVEYORS.GL11.PP_ENTER_OFF_TimerOff_Done_Bit;

// DE-BOUNCE TIMER FOR GL11 PP EXIT SWITCH ON
GVL_CONVEYORS.GL11.PP_EXIT_ON_TimerOn (IN := GVL_CONVEYORS.GL11.PP_EXIT_Left, PT := GVL_HMI.GL11PPExitOnPresetTime);
GVL_CONVEYORS.GL11.PP_EXIT_ON_TimerOn_Done_Bit := GVL_CONVEYORS.GL11.PP_EXIT_ON_TimerOn.Q;
GVL_CONVEYORS.GL11.PP_EXIT_ON_TimerOn_ELAPSED := GVL_CONVEYORS.GL11.PP_EXIT_ON_TimerOn.ET;
GVL_CONVEYORS.GL11.EXIT_SWITCH_IS_ON  := GVL_CONVEYORS.GL11.PP_EXIT_ON_TimerOn_Done_Bit;

// DE-BOUNCE TIMER FOR GL11 PP EXIT SWITCH OFF
GVL_CONVEYORS.GL11.PP_EXIT_OFF_TimerOff (IN := NOT GVL_CONVEYORS.GL11.PP_EXIT_left, PT := GVL_HMI.GL11PPExitOffPresetTime);
GVL_CONVEYORS.GL11.PP_EXIT_OFF_TimerOFF_Done_Bit := GVL_CONVEYORS.GL11.PP_EXIT_OFF_TimerOFF.Q;
GVL_CONVEYORS.GL11.PP_EXIT_OFF_TimerOFF_ELAPSED := GVL_CONVEYORS.GL11.PP_EXIT_OFF_TimerOFF.ET;
GVL_CONVEYORS.GL11.EXIT_SWITCH_IS_OFF  := GVL_CONVEYORS.GL11.PP_EXIT_OFF_TimerOff_Done_Bit;


// DE-BOUNCE TIMER FOR GL11 AT GL3 PROX 1 SWITCH ON
GVL_CONVEYORS.GL11.AT_GL3_PROX_1_ON_TimerOn (IN := GVL_CONVEYORS.GL11.At_GL3_Prox_1, PT := GVL_HMI.GL11ATGL3PositionProx1OnPresetTime);
GVL_CONVEYORS.GL11.AT_GL3_PROX_1_ON_TimerOn_Done_Bit := GVL_CONVEYORS.GL11.AT_GL3_PROX_1_ON_TimerOn.Q;
GVL_CONVEYORS.GL11.AT_GL3_PROX_1_ON_TimerOn_ELAPSED := GVL_CONVEYORS.GL11.AT_GL3_PROX_1_ON_TimerOn.ET;
GVL_CONVEYORS.GL11.AT_GL3_PROX_1_ON := GVL_CONVEYORS.GL11.AT_GL3_PROX_1_ON_TimerOn_Done_Bit;

// DE-BOUNCE TIMER FOR GL11 AT GL3 PROX 1 SWITCH OFF
GVL_CONVEYORS.GL11.AT_GL3_PROX_1_OFF_TimerOff (IN := NOT GVL_CONVEYORS.GL11.At_GL3_Prox_1, PT := GVL_HMI.GL11ATGL3PositionProx1OffPresetTime);
GVL_CONVEYORS.GL11.AT_GL3_PROX_1_OFF_TimerOFF_Done_Bit := GVL_CONVEYORS.GL11.AT_GL3_PROX_1_OFF_TimerOFF.Q;
GVL_CONVEYORS.GL11.AT_GL3_PROX_1_OFF_TimerOFF_ELAPSED := GVL_CONVEYORS.GL11.AT_GL3_PROX_1_OFF_TimerOFF.ET;
GVL_CONVEYORS.GL11.AT_GL3_PROX_1_OFF := GVL_CONVEYORS.GL11.AT_GL3_PROX_1_OFF_TimerOFF_Done_Bit;

// DE-BOUNCE TIMER FOR GL11 AT GL3 PROX 2 SWITCH ON
GVL_CONVEYORS.GL11.AT_GL3_PROX_2_ON_TimerOn (IN := GVL_CONVEYORS.GL11.At_GL3_Prox_2, PT := GVL_HMI.GL11ATGL3PositionProx2OnPresetTime);
GVL_CONVEYORS.GL11.AT_GL3_PROX_2_ON_TimerOn_Done_Bit := GVL_CONVEYORS.GL11.AT_GL3_PROX_2_ON_TimerOn.Q;
GVL_CONVEYORS.GL11.AT_GL3_PROX_2_ON_TimerOn_ELAPSED := GVL_CONVEYORS.GL11.AT_GL3_PROX_2_ON_TimerOn.ET;
GVL_CONVEYORS.GL11.AT_GL3_PROX_2_ON := GVL_CONVEYORS.GL11.AT_GL3_PROX_2_ON_TimerOn_Done_Bit;

// DE-BOUNCE TIMER FOR GL11 AT GL3 PROX 2 SWITCH OFF
GVL_CONVEYORS.GL11.AT_GL3_PROX_2_OFF_TimerOff (IN := NOT GVL_CONVEYORS.GL11.At_GL3_Prox_2, PT := GVL_HMI.GL11ATGL3PositionProx2OffPresetTime);
GVL_CONVEYORS.GL11.AT_GL3_PROX_2_OFF_TimerOFF_Done_Bit := GVL_CONVEYORS.GL11.AT_GL3_PROX_2_OFF_TimerOFF.Q;
GVL_CONVEYORS.GL11.AT_GL3_PROX_2_OFF_TimerOFF_ELAPSED := GVL_CONVEYORS.GL11.AT_GL3_PROX_2_OFF_TimerOFF.ET;
GVL_CONVEYORS.GL11.AT_GL3_PROX_2_OFF := GVL_CONVEYORS.GL11.AT_GL3_PROX_2_OFF_TimerOFF_Done_Bit;


// DE-BOUNCE TIMER FOR GL11 AT GL7 PROX 1 SWITCH ON
GVL_CONVEYORS.GL11.AT_GL7_PROX_1_ON_TimerOn (IN := GVL_CONVEYORS.GL11.At_GL7_Prox_1, PT := GVL_HMI.GL11ATGL7PositionProx1OnPresetTime);
GVL_CONVEYORS.GL11.AT_GL7_PROX_1_ON_TimerOn_Done_Bit := GVL_CONVEYORS.GL11.AT_GL7_PROX_1_ON_TimerOn.Q;
GVL_CONVEYORS.GL11.AT_GL7_PROX_1_ON_TimerOn_ELAPSED := GVL_CONVEYORS.GL11.AT_GL7_PROX_1_ON_TimerOn.ET;
GVL_CONVEYORS.GL11.AT_GL7_PROX_1_ON := GVL_CONVEYORS.GL11.AT_GL7_PROX_1_ON_TimerOn_Done_Bit;

// DE-BOUNCE TIMER FOR GL11 AT GL7 PROX 1 SWITCH OFF
GVL_CONVEYORS.GL11.AT_GL7_PROX_1_OFF_TimerOff (IN := NOT GVL_CONVEYORS.GL11.AT_GL7_PROX_1, PT := GVL_HMI.GL11ATGL7PositionProx1OffPresetTime);
GVL_CONVEYORS.GL11.AT_GL7_PROX_1_OFF_TimerOff_Done_Bit := GVL_CONVEYORS.GL11.AT_GL7_PROX_1_OFF_TimerOff.Q;
GVL_CONVEYORS.GL11.AT_GL7_PROX_1_OFF_TimerOff_ELAPSED := GVL_CONVEYORS.GL11.AT_GL7_PROX_1_OFF_TimerOff.ET;
GVL_CONVEYORS.GL11.AT_GL7_PROX_1_OFF := GVL_CONVEYORS.GL11.AT_GL7_PROX_1_OFF_TimerOff_Done_Bit;

// DE-BOUNCE TIMER FOR GL11 AT GL9 PROX 1 SWITCH ON
GVL_CONVEYORS.GL11.AT_GL9_PROX_1_ON_TimerOn (IN := GVL_CONVEYORS.GL11.At_GL9_Prox_1, PT := GVL_HMI.GL11ATGL9PositionProx1OnPresetTime);
GVL_CONVEYORS.GL11.AT_GL9_PROX_1_ON_TimerOn_Done_Bit:= GVL_CONVEYORS.GL11.AT_GL9_PROX_1_ON_TimerOn.Q;
GVL_CONVEYORS.GL11.AT_GL9_PROX_1_ON_TimerOn_ELAPSED := GVL_CONVEYORS.GL11.AT_GL9_PROX_1_ON_TimerOn.ET;
GVL_CONVEYORS.GL11.AT_GL9_PROX_1_ON := GVL_CONVEYORS.GL11.AT_GL9_PROX_1_ON_TimerOn_Done_Bit;

// DE-BOUNCE TIMER FOR GL11 AT GL9 PROX 1 SWITCH OFF
GVL_CONVEYORS.GL11.AT_GL9_Prox_1_OFF_TimerOff (IN := NOT GVL_CONVEYORS.GL11.AT_GL9_Prox_1, PT := GVL_HMI.GL11ATGL9PositionProx1OffPresetTime);
GVL_CONVEYORS.GL11.AT_GL9_Prox_1_OFF_TimerOff_Done_Bit := GVL_CONVEYORS.GL11.AT_GL9_Prox_1_OFF_TimerOff.Q;
GVL_CONVEYORS.GL11.AT_GL9_PROX_1_OFF_TimerOff_ELAPSED := GVL_CONVEYORS.GL11.AT_GL9_Prox_1_OFF_TimerOff.ET;
GVL_CONVEYORS.GL11.AT_GL9_Prox_1_OFF  := GVL_CONVEYORS.GL11.AT_GL9_Prox_1_OFF_TimerOff_Done_Bit;

// DE-BOUNCE TIMER FOR GL11 AT GL12 PROX 1 SWITCH ON
GVL_CONVEYORS.GL11.AT_GL12_PROX_1_ON_TimerOn (IN := GVL_CONVEYORS.GL11.AT_GL12_Prox_1, PT := GVL_HMI.GL11ATGL12PositionProx1OnPresetTime);
GVL_CONVEYORS.GL11.AT_GL12_PROX_1_ON_TimerOn_Done_Bit := GVL_CONVEYORS.GL11.AT_GL12_PROX_1_ON_TimerOn.Q;
GVL_CONVEYORS.GL11.AT_GL12_PROX_1_ON_TimerOn_ELAPSED := GVL_CONVEYORS.GL11.AT_GL12_PROX_1_ON_TimerOn.ET;
GVL_CONVEYORS.GL11.AT_GL12_PROX_1_ON := GVL_CONVEYORS.GL11.AT_GL12_PROX_1_ON_TimerOn_Done_Bit;

// DE-BOUNCE TIMER FOR GL11 AT GL12 PROX 1 SWITCH OFF
GVL_CONVEYORS.GL11.AT_GL12_PROX_1_OFF_TimerOff (IN := NOT GVL_CONVEYORS.GL11.AT_GL12_PROX_1, PT := GVL_HMI.GL11ATGL12PositionProx1OffPresetTime);
GVL_CONVEYORS.GL11.AT_GL12_PROX_1_OFF_TimerOff_Done_Bit := GVL_CONVEYORS.GL11.AT_GL12_PROX_1_OFF_TimerOff.Q;
GVL_CONVEYORS.GL11.AT_GL12_PROX_1_OFF_TimerOff_ELAPSED := GVL_CONVEYORS.GL11.AT_GL12_PROX_1_OFF_TimerOff.ET;
GVL_CONVEYORS.GL11.AT_GL12_PROX_1_OFF  := GVL_CONVEYORS.GL11.AT_GL12_PROX_1_OFF_TimerOff_Done_Bit;

// DE-BOUNCE TIMER FOR GL11 AT GL12 PROX 2 SWITCH ON
GVL_CONVEYORS.GL11.AT_GL12_PROX_2_ON_TimerOn (IN := GVL_CONVEYORS.GL11.AT_GL12_Prox_2, PT := GVL_HMI.GL11ATGL12PositionProx2OnPresetTime);
GVL_CONVEYORS.GL11.AT_GL12_PROX_2_ON_TimerOn_Done_Bit := GVL_CONVEYORS.GL11.AT_GL12_PROX_2_ON_TimerOn.Q;
GVL_CONVEYORS.GL11.AT_GL12_PROX_2_ON_TimerOn_ELAPSED := GVL_CONVEYORS.GL11.AT_GL12_PROX_2_ON_TimerOn.ET;
GVL_CONVEYORS.GL11.AT_GL12_PROX_2_ON := GVL_CONVEYORS.GL11.AT_GL12_PROX_2_ON_TimerOn_Done_Bit;

// DE-BOUNCE TIMER FOR GL11 AT GL12 PROX 2 SWITCH OFF
GVL_CONVEYORS.GL11.AT_GL12_PROX_2_OFF_TimerOff (IN := NOT GVL_CONVEYORS.GL11.AT_GL12_PROX_2, PT := GVL_HMI.GL11ATGL12PositionProx2OffPresetTime);
GVL_CONVEYORS.GL11.AT_GL12_PROX_2_OFF_TimerOff_Done_Bit := GVL_CONVEYORS.GL11.AT_GL12_PROX_2_OFF_TimerOff.Q;
GVL_CONVEYORS.GL11.AT_GL12_PROX_2_OFF_TimerOff_ELAPSED := GVL_CONVEYORS.GL11.AT_GL12_PROX_2_OFF_TimerOff.ET;
GVL_CONVEYORS.GL11.AT_GL12_PROX_2_OFF  := GVL_CONVEYORS.GL11.AT_GL12_PROX_2_OFF_TimerOff_Done_Bit;


// DE-BOUNCE TIMER FOR GL12 PP EXIT SWITCH ON
GVL_CONVEYORS.GL12.PP_EXIT_ON_TimerOn (IN := GVL_CONVEYORS.GL12.PP_EXIT_left, PT := GVL_HMI.GL12PPExitOnPresetTime);
GVL_CONVEYORS.GL12.PP_EXIT_ON_TimerOn_Done_Bit := GVL_CONVEYORS.GL12.PP_EXIT_ON_TimerOn.Q;
GVL_CONVEYORS.GL12.PP_EXIT_ON_TimerOn_ELAPSED := GVL_CONVEYORS.GL12.PP_EXIT_ON_TimerOn.ET;
GVL_CONVEYORS.GL12.EXIT_Switch_is_On  := GVL_CONVEYORS.GL12.PP_EXIT_ON_TimerOn_Done_Bit;

// DE-BOUNCE TIMER FOR GL12 PP EXIT SWITCH OFF
GVL_CONVEYORS.GL12.PP_EXIT_OFF_TimerOff (IN := NOT GVL_CONVEYORS.GL12.PP_EXIT_left, PT := GVL_HMI.GL12PPExitOffPresetTime);
GVL_CONVEYORS.GL12.PP_EXIT_OFF_TimerOFF_Done_Bit := GVL_CONVEYORS.GL12.PP_EXIT_OFF_TimerOFF.Q;
GVL_CONVEYORS.GL12.PP_EXIT_OFF_TimerOFF_ELAPSED := GVL_CONVEYORS.GL12.PP_EXIT_OFF_TimerOFF.ET;
GVL_CONVEYORS.GL12.Exit_Switch_is_Off  := GVL_CONVEYORS.GL12.PP_EXIT_OFF_TimerOff_Done_Bit;

// DE-BOUNCE TIMER FOR GL12 PP ENTER SWITCH ON
GVL_CONVEYORS.GL12.PP_ENTER_ON_TimerOn (IN := GVL_CONVEYORS.GL12.PP_ENTER_left, PT := GVL_HMI.GL12PPEnterOnPresetTime);
GVL_CONVEYORS.GL12.PP_ENTER_ON_TimerOn_Done_Bit := GVL_CONVEYORS.GL12.PP_ENTER_ON_TimerOn.Q;
GVL_CONVEYORS.GL12.PP_ENTER_ON_TimerOn_ELAPSED := GVL_CONVEYORS.GL12.PP_ENTER_ON_TimerOn.ET;
GVL_CONVEYORS.GL12.Enter_Switch_is_On  := GVL_CONVEYORS.GL12.PP_ENTER_ON_TimerOn_Done_Bit;

// DE-BOUNCE TIMER FOR GL12 PP ENTER SWITCH OFF
GVL_CONVEYORS.GL12.PP_ENTER_OFF_TimerOff (IN := NOT GVL_CONVEYORS.GL12.PP_ENTER_left, PT := GVL_HMI.GL12PPEnterOffPresetTime);
GVL_CONVEYORS.GL12.PP_ENTER_OFF_TimerOFF_Done_Bit := GVL_CONVEYORS.GL12.PP_ENTER_OFF_TimerOFF.Q;
GVL_CONVEYORS.GL12.PP_ENTER_OFF_TimerOFF_ELAPSED := GVL_CONVEYORS.GL12.PP_ENTER_OFF_TimerOFF.ET;
GVL_CONVEYORS.GL12.Enter_Switch_is_Off  := GVL_CONVEYORS.GL12.PP_ENTER_OFF_TimerOff_Done_Bit;


///////////////////////////////////////ROLL UP DOORS//////////////////////////////////////////

//DE-BOUNCE TIMER FOR GL1 ROLL DOOR UP SWITCH ON
GVL_CONVEYORS.GL1_RD.DOOR_IS_UP_TimerOn (IN := GVL_CONVEYORS.GL1_Rd.DOOR_OPEN_SWITCH, PT := T#500MS);
GVL_CONVEYORS.GL1_RD.DOOR_IS_UP_TimerOn_Done_Bit := GVL_CONVEYORS.GL1_RD.DOOR_IS_UP_TimerOn.Q;
GVL_CONVEYORS.GL1_RD.DOOR_IS_UP_TIMER_ON_ELAPSED := GVL_CONVEYORS.GL1_RD.DOOR_IS_UP_TimerOn.ET;
GVL_CONVEYORS.GL1_RD.UP_SWITCH_IS_ON:= GVL_CONVEYORS.GL1_RD.DOOR_IS_UP_TimerOn_Done_Bit;

// DE-BOUNCE TIMER FOR GL1 ROLL DOOR UP SWITCH OFF
GVL_CONVEYORS.GL1_RD.DOOR_IS_UP_TimerOFF (IN := NOT GVL_CONVEYORS.GL1_RD.DOOR_OPEN_SWITCH, PT := T#500MS);
GVL_CONVEYORS.GL1_RD.DOOR_IS_UP_TimerOFF_Done_Bit := GVL_CONVEYORS.GL1_RD.DOOR_IS_UP_TimerOff.Q;
GVL_CONVEYORS.GL1_RD.DOOR_IS_UP_TIMER_OFF_ELAPSED := GVL_CONVEYORS.GL1_RD.DOOR_IS_UP_TimerOff.ET;
GVL_CONVEYORS.GL1_RD.UP_SWITCH_IS_ON:= GVL_CONVEYORS.GL1_RD.DOOR_IS_UP_TimerOn_Done_Bit;

// DE-BOUNCE TIMER FOR GL1 ROLL DOOR DOWN SWITCH ON
GVL_CONVEYORS.GL1_RD.DOOR_IS_DOWN_TimerOn (IN := GVL_CONVEYORS.GL1_RD.DOOR_CLOSED_SWITCH, PT := T#500MS);
GVL_CONVEYORS.GL1_RD.DOOR_IS_DOWN_TimerOn_Done_Bit := GVL_CONVEYORS.GL1_RD.DOOR_IS_DOWN_TimerOn.Q;
GVL_CONVEYORS.GL1_RD.DOOR_IS_DOWN_TIMER_ON_ELAPSED := GVL_CONVEYORS.GL1_RD.DOOR_IS_DOWN_TimerOn.ET;
GVL_CONVEYORS.GL1_RD.DOWN_SWITCH_IS_ON := GVL_CONVEYORS.GL1_RD.DOOR_IS_DOWN_TimerOn_Done_Bit;

// DE-BOUNCE TIMER FOR GL1 ROLL DOOR DOWN SWITCH OFF
GVL_CONVEYORS.GL1_RD.DOOR_IS_DOWN_TimerOFF (IN := NOT GVL_CONVEYORS.GL1_RD.DOOR_CLOSED_SWITCH, PT := T#500MS);
GVL_CONVEYORS.GL1_RD.DOOR_IS_DOWN_TimerOFF_Done_Bit := GVL_CONVEYORS.GL1_RD.DOOR_IS_DOWN_TimerOff.Q;
GVL_CONVEYORS.GL1_RD.DOOR_IS_DOWN_TIMER_OFF_ELAPSED := GVL_CONVEYORS.GL1_RD.DOOR_IS_DOWN_TimerOff.ET;
GVL_CONVEYORS.GL1_RD.DOWN_SWITCH_IS_OFF := GVL_CONVEYORS.GL1_RD.DOOR_IS_DOWN_TimerOFF_Done_Bit;

//DE-BOUNCE TIMER FOR GL6 ROLL DOOR UP SWITCH ON
GVL_CONVEYORS.GL6_RD.DOOR_IS_UP_TimerOn (IN := GVL_CONVEYORS.GL6_Rd.DOOR_OPEN_SWITCH, PT := T#500MS);
GVL_CONVEYORS.GL6_RD.DOOR_IS_UP_TimerOn_Done_Bit := GVL_CONVEYORS.GL6_RD.DOOR_IS_UP_TimerOn.Q;
GVL_CONVEYORS.GL6_RD.DOOR_IS_UP_TIMER_ON_ELAPSED := GVL_CONVEYORS.GL6_RD.DOOR_IS_UP_TimerOn.ET;
GVL_CONVEYORS.GL6_RD.UP_SWITCH_IS_ON:= GVL_CONVEYORS.GL6_RD.DOOR_IS_UP_TimerOn_Done_Bit;

// DE-BOUNCE TIMER FOR GL6 ROLL DOOR UP SWITCH OFF
GVL_CONVEYORS.GL6_RD.DOOR_IS_UP_TimerOFF (IN := NOT GVL_CONVEYORS.GL6_RD.DOOR_OPEN_SWITCH, PT := T#500MS);
GVL_CONVEYORS.GL6_RD.DOOR_IS_UP_TimerOFF_Done_Bit := GVL_CONVEYORS.GL6_RD.DOOR_IS_UP_TimerOff.Q;
GVL_CONVEYORS.GL6_RD.DOOR_IS_UP_TIMER_OFF_ELAPSED := GVL_CONVEYORS.GL6_RD.DOOR_IS_UP_TimerOff.ET;
GVL_CONVEYORS.GL6_RD.UP_SWITCH_IS_ON:= GVL_CONVEYORS.GL6_RD.DOOR_IS_UP_TimerOn_Done_Bit;

// DE-BOUNCE TIMER FOR GL6 ROLL DOOR DOWN SWITCH ON
GVL_CONVEYORS.GL1_RD.DOOR_IS_DOWN_TimerOn (IN := GVL_CONVEYORS.GL1_RD.DOOR_CLOSED_SWITCH, PT := T#500MS);
GVL_CONVEYORS.GL1_RD.DOOR_IS_DOWN_TimerOn_Done_Bit := GVL_CONVEYORS.GL1_RD.DOOR_IS_DOWN_TimerOn.Q;
GVL_CONVEYORS.GL1_RD.DOOR_IS_DOWN_TIMER_ON_ELAPSED := GVL_CONVEYORS.GL1_RD.DOOR_IS_DOWN_TimerOn.ET;
GVL_CONVEYORS.GL1_RD.DOWN_SWITCH_IS_ON := GVL_CONVEYORS.GL1_RD.DOOR_IS_DOWN_TimerOn_Done_Bit;

// DE-BOUNCE TIMER FOR GL6 ROLL DOOR DOWN SWITCH OFF
GVL_CONVEYORS.GL6_RD.DOOR_IS_DOWN_TimerOFF (IN := NOT GVL_CONVEYORS.GL6_RD.DOOR_CLOSED_SWITCH, PT := T#500MS);
GVL_CONVEYORS.GL6_RD.DOOR_IS_DOWN_TimerOFF_Done_Bit := GVL_CONVEYORS.GL6_RD.DOOR_IS_DOWN_TimerOff.Q;
GVL_CONVEYORS.GL6_RD.DOOR_IS_DOWN_TIMER_OFF_ELAPSED := GVL_CONVEYORS.GL6_RD.DOOR_IS_DOWN_TimerOff.ET;
GVL_CONVEYORS.GL6_RD.DOWN_SWITCH_IS_OFF := GVL_CONVEYORS.GL6_RD.DOOR_IS_DOWN_TimerOFF_Done_Bit;

// DE-BOUNCE TIMER FOR GL8 ROLL DOOR UP SWITCH OFF
GVL_CONVEYORS.GL6_RD.DOOR_IS_UP_TimerOFF (IN := NOT GVL_CONVEYORS.GL6_RD.DOOR_OPEN_SWITCH, PT := T#500MS);
GVL_CONVEYORS.GL6_RD.DOOR_IS_UP_TimerOFF_Done_Bit := GVL_CONVEYORS.GL6_RD.DOOR_IS_UP_TimerOff.Q;
GVL_CONVEYORS.GL6_RD.DOOR_IS_UP_TIMER_OFF_ELAPSED := GVL_CONVEYORS.GL6_RD.DOOR_IS_UP_TimerOff.ET;
GVL_CONVEYORS.GL6_RD.UP_SWITCH_IS_ON:= GVL_CONVEYORS.GL6_RD.DOOR_IS_UP_TimerOn_Done_Bit;

//DE-BOUNCE TIMER FOR GL8 ROLL DOOR UP SWITCH ON
GVL_CONVEYORS.GL8_RD.DOOR_IS_UP_TimerOn (IN := GVL_CONVEYORS.GL8_Rd.DOOR_OPEN_SWITCH, PT := T#500MS);
GVL_CONVEYORS.GL8_RD.DOOR_IS_UP_TimerOn_Done_Bit := GVL_CONVEYORS.GL8_RD.DOOR_IS_UP_TimerOn.Q;
GVL_CONVEYORS.GL8_RD.DOOR_IS_UP_TIMER_ON_ELAPSED := GVL_CONVEYORS.GL8_RD.DOOR_IS_UP_TimerOn.ET;
GVL_CONVEYORS.GL8_RD.UP_SWITCH_IS_ON:= GVL_CONVEYORS.GL8_RD.DOOR_IS_UP_TimerOn_Done_Bit;

// DE-BOUNCE TIMER FOR GL8 ROLL DOOR DOWN SWITCH ON
GVL_CONVEYORS.GL8_RD.DOOR_IS_DOWN_TimerOn (IN := GVL_CONVEYORS.GL8_RD.DOOR_CLOSED_SWITCH, PT := T#500MS);
GVL_CONVEYORS.GL8_RD.DOOR_IS_DOWN_TimerOn_Done_Bit := GVL_CONVEYORS.GL8_RD.DOOR_IS_DOWN_TimerOn.Q;
GVL_CONVEYORS.GL8_RD.DOOR_IS_DOWN_TIMER_ON_ELAPSED := GVL_CONVEYORS.GL8_RD.DOOR_IS_DOWN_TimerOn.ET;
GVL_CONVEYORS.GL8_RD.DOWN_SWITCH_IS_ON := GVL_CONVEYORS.GL8_RD.DOOR_IS_DOWN_TimerOn_Done_Bit;

// DE-BOUNCE TIMER FOR GL8 ROLL DOOR DOWN SWITCH OFF
GVL_CONVEYORS.GL8_RD.DOOR_IS_DOWN_TimerOFF (IN := NOT GVL_CONVEYORS.GL8_RD.DOOR_CLOSED_SWITCH, PT := T#500MS);
GVL_CONVEYORS.GL8_RD.DOOR_IS_DOWN_TimerOFF_Done_Bit := GVL_CONVEYORS.GL8_RD.DOOR_IS_DOWN_TimerOFF.Q;
GVL_CONVEYORS.GL8_RD.DOOR_IS_DOWN_TIMER_OFF_ELAPSED := GVL_CONVEYORS.GL8_RD.DOOR_IS_DOWN_TimerOff.ET;
GVL_CONVEYORS.GL8_RD.DOWN_SWITCH_IS_OFF := GVL_CONVEYORS.GL8_RD.DOOR_IS_DOWN_TimerOFF_Done_Bit;

///// CASE STOPS RAISE/LOWER SWITCHES

// DE-BOUNCE TIMER FOR GL2 CASE STOP IS RAISED SWITCH ON
GVL_CONVEYORS.GL2.CaseStopIsRaisedTimerOn (IN := GVL_CONVEYORS.GL2.Case_Stop_Extended_Right AND GVL_CONVEYORS.GL2.Case_Stop_Extended_Left , PT := T#500MS);
GVL_CONVEYORS.GL2.CaseStopIsRaisedTimerOnDoneBit := GVL_CONVEYORS.GL2.CaseStopIsRaisedTimerOn.Q;
GVL_CONVEYORS.GL2.CaseStopIsRaisedTimerOnElapsedTime := GVL_CONVEYORS.GL2.CaseStopIsRaisedTimerOn.ET;
GVL_CONVEYORS.GL2.CaseStopRaisedSwitchIsOn := GVL_CONVEYORS.GL2.CaseStopIsRaisedTimerOnDoneBit;

//// DE-BOUNCE TIMER FOR GL2 CASE STOP IS RAISED SWITCH OFF
GVL_CONVEYORS.GL2.CaseStopIsRaisedTimerOff (IN := GVL_CONVEYORS.GL2.Case_Stop_Extended_Right AND GVL_CONVEYORS.GL2.Case_Stop_Extended_Left , PT := T#500MS);
GVL_CONVEYORS.GL2.CaseStopIsRaisedTimerOffDoneBit := GVL_CONVEYORS.GL2.CaseStopIsRaisedTimerOff.Q;
GVL_CONVEYORS.GL2.CaseStopIsRaisedTimerOffElapsedTime := GVL_CONVEYORS.GL2.CaseStopIsRaisedTimerOff.ET;
GVL_CONVEYORS.GL2.CaseStopRaisedSwitchIsOff := GVL_CONVEYORS.GL2.CaseStopIsRaisedTimerOffDoneBit;

//// DE-BOUNCE TIMER FOR GL2 CASE STOP IS LOWERED SWITCH ON
GVL_CONVEYORS.GL2.CaseStopIsLoweredTimerOn (IN := GVL_CONVEYORS.GL2.Case_Stop_Retracted_Right AND GVL_CONVEYORS.GL2.Case_Stop_Retracted_Left , PT := T#500MS);
GVL_CONVEYORS.GL2.CaseStopIsLoweredTimerOnDoneBit := GVL_CONVEYORS.GL2.CaseStopIsLoweredTimerOn.Q;
GVL_CONVEYORS.GL2.CaseStopIsLoweredTimerOnElapsedTime := GVL_CONVEYORS.GL2.CaseStopIsLoweredTimerOn.ET;
GVL_CONVEYORS.GL2.CaseStopLoweredSwitchIsOn := GVL_CONVEYORS.GL2.CaseStopIsLoweredTimerOnDoneBit;

// DE-BOUNCE TIMER FOR GL2 CASE STOP IS LOWERED SWITCH OFF
GVL_CONVEYORS.GL2.CaseStopIsLoweredTimerOff (IN := GVL_CONVEYORS.GL2.Case_Stop_Retracted_Right AND GVL_CONVEYORS.GL2.Case_Stop_Retracted_Left , PT := T#500MS);
GVL_CONVEYORS.GL2.CaseStopIsLoweredTimerOffDoneBit := GVL_CONVEYORS.GL2.CaseStopIsLoweredTimerOff.Q;
GVL_CONVEYORS.GL2.CaseStopIsLoweredTimerOffElapsedTime := GVL_CONVEYORS.GL2.CaseStopIsLoweredTimerOff.ET;
GVL_CONVEYORS.GL2.CaseStopLoweredSwitchIsOff := GVL_CONVEYORS.GL2.CaseStopIsLoweredTimerOffDoneBit;

// DE-BOUNCE TIMER FOR GL3 CASE STOP IS LOWERED SWITCH ON
GVL_CONVEYORS.GL3.CaseStopIsLoweredTimerOn (IN := GVL_CONVEYORS.GL3.Case_Stop_Retracted_Right AND GVL_CONVEYORS.GL3.Case_Stop_Retracted_Left , PT := T#500MS);
GVL_CONVEYORS.GL3.CaseStopIsLoweredTimerOnDoneBit := GVL_CONVEYORS.GL3.CaseStopIsLoweredTimerOn.Q;
GVL_CONVEYORS.GL3.CaseStopIsLoweredTimerOnElapsedTime := GVL_CONVEYORS.GL3.CaseStopIsLoweredTimerOn.ET;
GVL_CONVEYORS.GL3.CaseStopLoweredSwitchIsOn := GVL_CONVEYORS.GL3.CaseStopIsLoweredTimerOnDoneBit;

// DE-BOUNCE TIMER FOR GL3 CASE STOP IS LOWERED SWITCH OFF
GVL_CONVEYORS.GL3.CaseStopIsLoweredTimerOff (IN := GVL_CONVEYORS.GL3.Case_Stop_Retracted_Right AND GVL_CONVEYORS.GL3.Case_Stop_Retracted_Left , PT := T#500MS);
GVL_CONVEYORS.GL3.CaseStopIsLoweredTimerOffDoneBit := GVL_CONVEYORS.GL3.CaseStopIsLoweredTimerOff.Q;
GVL_CONVEYORS.GL3.CaseStopIsLoweredTimerOffElapsedTime := GVL_CONVEYORS.GL3.CaseStopIsLoweredTimerOff.ET;
GVL_CONVEYORS.GL3.CaseStopLoweredSwitchIsOff := GVL_CONVEYORS.GL3.CaseStopIsLoweredTimerOffDoneBit;

// DE-BOUNCE TIMER FOR GL3 CASE STOP IS RAISED SWITCH ON
GVL_CONVEYORS.GL3.CaseStopIsRaisedTimerOn (IN := GVL_CONVEYORS.GL3.Case_Stop_Extended_Right AND GVL_CONVEYORS.GL3.Case_Stop_Extended_Left , PT := T#500MS);
GVL_CONVEYORS.GL3.CaseStopIsRaisedTimerOnDoneBit := GVL_CONVEYORS.GL3.CaseStopIsRaisedTimerOn.Q;
GVL_CONVEYORS.GL3.CaseStopIsRaisedTimerOnElapsedTime := GVL_CONVEYORS.GL3.CaseStopIsRaisedTimerOn.ET;
GVL_CONVEYORS.GL3.CaseStopRaisedSwitchIsOn := GVL_CONVEYORS.GL3.CaseStopIsRaisedTimerOnDoneBit;

// DE-BOUNCE TIMER FOR GL3 CASE STOP IS RAISED SWITCH OFF
GVL_CONVEYORS.GL4.CaseStopIsRaisedTimerOff (IN := GVL_CONVEYORS.GL4.Case_Stop_Extended_Right AND GVL_CONVEYORS.GL4.Case_Stop_Extended_Left , PT := T#500MS);
GVL_CONVEYORS.GL4.CaseStopIsRaisedTimerOffDoneBit := GVL_CONVEYORS.GL4.CaseStopIsRaisedTimerOff.Q;
GVL_CONVEYORS.GL4.CaseStopIsRaisedTimerOffElapsedTime := GVL_CONVEYORS.GL4.CaseStopIsRaisedTimerOff.ET;
GVL_CONVEYORS.GL4.CaseStopRaisedSwitchIsOff := GVL_CONVEYORS.GL4.CaseStopIsRaisedTimerOffDoneBit;


// DE-BOUNCE TIMER FOR GL4 CASE STOP IS LOWERED SWITCH ON
GVL_CONVEYORS.GL4.CaseStopIsLoweredTimerOn (IN := GVL_CONVEYORS.GL4.Case_Stop_Retracted_Right AND GVL_CONVEYORS.GL4.Case_Stop_Retracted_Left , PT := T#500MS);
GVL_CONVEYORS.GL4.CaseStopIsLoweredTimerOnDoneBit := GVL_CONVEYORS.GL4.CaseStopIsLoweredTimerOn.Q;
GVL_CONVEYORS.GL4.CaseStopIsLoweredTimerOnElapsedTime := GVL_CONVEYORS.GL4.CaseStopIsLoweredTimerOn.ET;
GVL_CONVEYORS.GL4.CaseStopLoweredSwitchIsOn := GVL_CONVEYORS.GL4.CaseStopIsLoweredTimerOnDoneBit;

// DE-BOUNCE TIMER FOR GL4 CASE STOP IS LOWERED SWITCH OFF
GVL_CONVEYORS.GL4.CaseStopIsLoweredTimerOff (IN := GVL_CONVEYORS.GL4.Case_Stop_Retracted_Right AND GVL_CONVEYORS.GL4.Case_Stop_Retracted_Left , PT := T#500MS);
GVL_CONVEYORS.GL4.CaseStopIsLoweredTimerOffDoneBit := GVL_CONVEYORS.GL4.CaseStopIsLoweredTimerOff.Q;
GVL_CONVEYORS.GL4.CaseStopIsLoweredTimerOffElapsedTime := GVL_CONVEYORS.GL4.CaseStopIsLoweredTimerOff.ET;
GVL_CONVEYORS.GL4.CaseStopLoweredSwitchIsOff := GVL_CONVEYORS.GL4.CaseStopIsLoweredTimerOffDoneBit;

// DE-BOUNCE TIMER FOR GL4 CASE STOP IS RAISED SWITCH ON
GVL_CONVEYORS.GL4.CaseStopIsRaisedTimerOn (IN := GVL_CONVEYORS.GL4.Case_Stop_Extended_Right AND GVL_CONVEYORS.GL4.Case_Stop_Extended_Left , PT := T#500MS);
GVL_CONVEYORS.GL4.CaseStopIsRaisedTimerOnDoneBit := GVL_CONVEYORS.GL4.CaseStopIsRaisedTimerOn.Q;
GVL_CONVEYORS.GL4.CaseStopIsRaisedTimerOnElapsedTime := GVL_CONVEYORS.GL4.CaseStopIsRaisedTimerOn.ET;
GVL_CONVEYORS.GL4.CaseStopRaisedSwitchIsOn := GVL_CONVEYORS.GL4.CaseStopIsRaisedTimerOnDoneBit;

// DE-BOUNCE TIMER FOR GL4 CASE STOP IS RAISED SWITCH OFF
GVL_CONVEYORS.GL4.CaseStopIsRaisedTimerOff (IN := GVL_CONVEYORS.GL4.Case_Stop_Extended_Right AND GVL_CONVEYORS.GL4.Case_Stop_Extended_Left , PT := T#500MS);
GVL_CONVEYORS.GL4.CaseStopIsRaisedTimerOffDoneBit := GVL_CONVEYORS.GL4.CaseStopIsRaisedTimerOff.Q;
GVL_CONVEYORS.GL4.CaseStopIsRaisedTimerOffElapsedTime := GVL_CONVEYORS.GL4.CaseStopIsRaisedTimerOff.ET;
GVL_CONVEYORS.GL4.CaseStopRaisedSwitchIsOff := GVL_CONVEYORS.GL4.CaseStopIsRaisedTimerOffDoneBit;

// DE-BOUNCE TIMER FOR GL5A CASE STOP IS LOWERED SWITCH ON
GVL_CONVEYORS.GL5A.CaseStopIsLoweredTimerOn (IN := GVL_CONVEYORS.GL5A.Case_Stop_Retracted_Right AND GVL_CONVEYORS.GL5A.Case_Stop_Retracted_Left , PT := T#500MS);
GVL_CONVEYORS.GL5A.CaseStopIsLoweredTimerOnDoneBit := GVL_CONVEYORS.GL5A.CaseStopIsLoweredTimerOn.Q;
GVL_CONVEYORS.GL5A.CaseStopIsLoweredTimerOnElapsedTime := GVL_CONVEYORS.GL5A.CaseStopIsLoweredTimerOn.ET;
GVL_CONVEYORS.GL5A.CaseStopLoweredSwitchIsOn := GVL_CONVEYORS.GL5A.CaseStopIsLoweredTimerOnDoneBit;

// DE-BOUNCE TIMER FOR GL5A CASE STOP IS LOWERED SWITCH OFF
GVL_CONVEYORS.GL5A.CaseStopIsLoweredTimerOff (IN := GVL_CONVEYORS.GL5A.Case_Stop_Retracted_Right AND GVL_CONVEYORS.GL5A.Case_Stop_Retracted_Left , PT := T#500MS);
GVL_CONVEYORS.GL5A.CaseStopIsLoweredTimerOffDoneBit := GVL_CONVEYORS.GL5A.CaseStopIsLoweredTimerOff.Q;
GVL_CONVEYORS.GL5A.CaseStopIsLoweredTimerOffElapsedTime := GVL_CONVEYORS.GL5A.CaseStopIsLoweredTimerOff.ET;
GVL_CONVEYORS.GL5A.CaseStopLoweredSwitchIsOff := GVL_CONVEYORS.GL5A.CaseStopIsLoweredTimerOffDoneBit;

// DE-BOUNCE TIMER FOR GL5A CASE STOP IS RAISED SWITCH ON
GVL_CONVEYORS.GL5A.CaseStopIsRaisedTimerOn (IN := GVL_CONVEYORS.GL5A.Case_Stop_Extended_Right AND GVL_CONVEYORS.GL5A.Case_Stop_Extended_Left , PT := T#500MS);
GVL_CONVEYORS.GL5A.CaseStopIsRaisedTimerOnDoneBit := GVL_CONVEYORS.GL5A.CaseStopIsRaisedTimerOn.Q;
GVL_CONVEYORS.GL5A.CaseStopIsRaisedTimerOnElapsedTime := GVL_CONVEYORS.GL5A.CaseStopIsRaisedTimerOn.ET;
GVL_CONVEYORS.GL5A.CaseStopRaisedSwitchIsOn := GVL_CONVEYORS.GL5A.CaseStopIsRaisedTimerOnDoneBit;

// DE-BOUNCE TIMER FOR GL5A CASE STOP IS RAISED SWITCH OFF
GVL_CONVEYORS.GL5A.CaseStopIsRaisedTimerOff (IN := GVL_CONVEYORS.GL5A.Case_Stop_Extended_Right AND GVL_CONVEYORS.GL5A.Case_Stop_Extended_Left , PT := T#500MS);
GVL_CONVEYORS.GL5A.CaseStopIsRaisedTimerOffDoneBit := GVL_CONVEYORS.GL5A.CaseStopIsRaisedTimerOff.Q;
GVL_CONVEYORS.GL5A.CaseStopIsRaisedTimerOffElapsedTime := GVL_CONVEYORS.GL5A.CaseStopIsRaisedTimerOff.ET;
GVL_CONVEYORS.GL5A.CaseStopRaisedSwitchIsOff := GVL_CONVEYORS.GL5A.CaseStopIsRaisedTimerOffDoneBit;


/////// DUAL CASE STOPS AT GL6 AND GL8
// DE-BOUNCE TIMER FOR GL6 CASE STOP1 IS LOWERED SWITCH ON
GVL_CONVEYORS.GL6.CaseStop1IsLoweredTimerOn (IN := GVL_CONVEYORS.GL6.Case_Stop_Load_1_Retracted_Right AND GVL_CONVEYORS.GL6.Case_Stop_Load_1_Retracted_Left , PT := T#500MS);
GVL_CONVEYORS.GL6.CaseStop1IsLoweredTimerOnDoneBit := GVL_CONVEYORS.GL6.CaseStop1IsLoweredTimerOn.Q;
GVL_CONVEYORS.GL6.CaseStop1IsLoweredTimerOnElapsedTime := GVL_CONVEYORS.GL6.CaseStop1IsLoweredTimerOn.ET;
GVL_CONVEYORS.GL6.CaseStop1LoweredSwitchIsOn := GVL_CONVEYORS.GL6.CaseStop1IsLoweredTimerOnDoneBit;

// DE-BOUNCE TIMER FOR GL6 CASE STOP1 IS LOWERED SWITCH OFF
GVL_CONVEYORS.GL6.CaseStop1IsLoweredTimerOFF (IN := GVL_CONVEYORS.GL6.Case_Stop_Load_1_Retracted_Right AND GVL_CONVEYORS.GL6.Case_Stop_Load_1_Retracted_Left , PT := T#500MS);
GVL_CONVEYORS.GL6.CaseStop1IsLoweredTimerOffDoneBit := GVL_CONVEYORS.GL5B.CaseStopIsLoweredTimerOff.Q;
GVL_CONVEYORS.GL6.CaseStop1IsLoweredTimerOffElapsedTime := GVL_CONVEYORS.GL5B.CaseStopIsLoweredTimerOff.ET;
GVL_CONVEYORS.GL6.CaseStop1LoweredSwitchIsOff := GVL_CONVEYORS.GL6.CaseStop1IsLoweredTimerOffDoneBit;

// DE-BOUNCE TIMER FOR GL6 CASE STOP1 IS RAISED SWITCH ON
GVL_CONVEYORS.GL6.CaseStop1IsRaisedTimerOn (IN := GVL_CONVEYORS.GL6.Case_Stop_Load_1_Extended_Right AND GVL_CONVEYORS.GL6.Case_Stop_Load_1_Extended_Left , PT := T#500MS);
GVL_CONVEYORS.GL6.CaseStop1IsRaisedTimerOnDoneBit := GVL_CONVEYORS.GL6.CaseStop1IsRaisedTimerOn.Q;
GVL_CONVEYORS.GL6.CaseStop1IsRaisedTimerOnElapsedTime := GVL_CONVEYORS.GL6.CaseStop1IsRaisedTimerOn.ET;
GVL_CONVEYORS.GL6.CaseStop1RaisedSwitchIsOn := GVL_CONVEYORS.GL6.CaseStop1IsRaisedTimerOnDoneBit;

// DE-BOUNCE TIMER FOR GL6 CASE STOP1 IS RAISED SWITCH OFF
GVL_CONVEYORS.GL6.CaseStop1IsRaisedTimerOff (IN := GVL_CONVEYORS.GL6.Case_Stop_Load_1_Extended_Right AND GVL_CONVEYORS.GL6.Case_Stop_Load_1_Extended_Left , PT := T#500MS);
GVL_CONVEYORS.GL6.CaseStop1IsRaisedTimerOffDoneBit := GVL_CONVEYORS.GL6.CaseStop1IsRaisedTimerOff.Q;
GVL_CONVEYORS.GL6.CaseStop1IsRaisedTimerOffElapsedTime := GVL_CONVEYORS.GL6.CaseStop1IsRaisedTimerOff.ET;
GVL_CONVEYORS.GL6.CaseStop1RaisedSwitchIsOff := GVL_CONVEYORS.GL6.CaseStop1IsRaisedTimerOffDoneBit;

// DE-BOUNCE TIMER FOR GL6 CASE STOP2 IS LOWERED SWITCH ON
GVL_CONVEYORS.GL6.CaseStop2IsLoweredTimerOn (IN := GVL_CONVEYORS.GL6.Case_Stop_Load_2_Retracted_Right AND GVL_CONVEYORS.GL6.Case_Stop_Load_2_Retracted_Left , PT := T#500MS);
GVL_CONVEYORS.GL6.CaseStop2IsLoweredTimerOnDoneBit := GVL_CONVEYORS.GL6.CaseStop2IsLoweredTimerOn.Q;
GVL_CONVEYORS.GL6.CaseStop2IsLoweredTimerOnElapsedTime := GVL_CONVEYORS.GL6.CaseStop2IsLoweredTimerOn.ET;
GVL_CONVEYORS.GL6.CaseStop2LoweredSwitchIsOn := GVL_CONVEYORS.GL6.CaseStop2IsLoweredTimerOnDoneBit;

// DE-BOUNCE TIMER FOR GL6 CASE STOP2 IS LOWERED SWITCH OFF
GVL_CONVEYORS.GL6.CaseStop2IsLoweredTimerOFF (IN := GVL_CONVEYORS.GL6.Case_Stop_Load_2_Retracted_Right AND GVL_CONVEYORS.GL6.Case_Stop_Load_2_Retracted_Left , PT := T#500MS);
GVL_CONVEYORS.GL6.CaseStopIsLoweredTimerOffDoneBit := GVL_CONVEYORS.GL6.CaseStop2IsLoweredTimerOff.Q;
GVL_CONVEYORS.GL6.CaseStop2IsLoweredTimerOffElapsedTime := GVL_CONVEYORS.GL6.CaseStop2IsLoweredTimerOff.ET;
GVL_CONVEYORS.GL6.CaseStop2LoweredSwitchIsOff := GVL_CONVEYORS.GL6.CaseStop2IsLoweredTimerOffDoneBit;

// DE-BOUNCE TIMER FOR GL6 CASE STOP2 IS RAISED SWITCH ON
GVL_CONVEYORS.GL6.CaseStop2IsRaisedTimerOn (IN := GVL_CONVEYORS.GL6.Case_Stop_Load_2_Extended_Right AND GVL_CONVEYORS.GL6.Case_Stop_Load_2_Extended_Left , PT := T#500MS);
GVL_CONVEYORS.GL6.CaseStop2IsRaisedTimerOnDoneBit := GVL_CONVEYORS.GL6.CaseStop2IsRaisedTimerOn.Q;
GVL_CONVEYORS.GL6.CaseStop2IsRaisedTimerOnElapsedTime := GVL_CONVEYORS.GL6.CaseStop2IsRaisedTimerOn.ET;
GVL_CONVEYORS.GL5B.CaseStopRaisedSwitchIsOn := GVL_CONVEYORS.GL5B.CaseStopIsRaisedTimerOnDoneBit;

// DE-BOUNCE TIMER FOR GL6 CASE STOP2 IS RAISED SWITCH OFF
GVL_CONVEYORS.GL6.CaseStop2IsRaisedTimerOff (IN := GVL_CONVEYORS.GL6.Case_Stop_Load_2_Extended_Right AND GVL_CONVEYORS.GL6.Case_Stop_Load_2_Extended_Left , PT := T#500MS);
GVL_CONVEYORS.GL6.CaseStop2IsRaisedTimerOffDoneBit := GVL_CONVEYORS.GL6.CaseStop2IsRaisedTimerOff.Q;
GVL_CONVEYORS.GL6.CaseStop2IsRaisedTimerOffElapsedTime := GVL_CONVEYORS.GL6.CaseStop2IsRaisedTimerOff.ET;
GVL_CONVEYORS.GL6.CaseStop2RaisedSwitchIsOff := GVL_CONVEYORS.GL6.CaseStop2IsRaisedTimerOffDoneBit;





// GL8 DUAL CASE STOPS
// DE-BOUNCE TIMER FOR GL8 CASE STOP1 IS LOWERED SWITCH ON
GVL_CONVEYORS.GL8.CaseStop1IsLoweredTimerOn (IN := GVL_CONVEYORS.GL8.Case_Stop_Load_1_Retracted_Right AND GVL_CONVEYORS.GL8.Case_Stop_Load_1_Retracted_Left , PT := T#500MS);
GVL_CONVEYORS.GL8.CaseStop1IsLoweredTimerOnDoneBit := GVL_CONVEYORS.GL8.CaseStop1IsLoweredTimerOn.Q;
GVL_CONVEYORS.GL8.CaseStop1IsLoweredTimerOnElapsedTime := GVL_CONVEYORS.GL8.CaseStop1IsLoweredTimerOn.ET;
GVL_CONVEYORS.GL8.CaseStop1LoweredSwitchIsOn := GVL_CONVEYORS.GL8.CaseStop1IsLoweredTimerOnDoneBit;

// DE-BOUNCE TIMER FOR GL8 CASE STOP1 IS LOWERED SWITCH OFF
GVL_CONVEYORS.GL8.CaseStop1IsLoweredTimerOFF (IN := GVL_CONVEYORS.GL8.Case_Stop_Load_1_Retracted_Right AND GVL_CONVEYORS.GL8.Case_Stop_Load_1_Retracted_Left , PT := T#500MS);
GVL_CONVEYORS.GL8.CaseStop1IsLoweredTimerOffDoneBit := GVL_CONVEYORS.GL5B.CaseStopIsLoweredTimerOff.Q;
GVL_CONVEYORS.GL8.CaseStop1IsLoweredTimerOffElapsedTime := GVL_CONVEYORS.GL5B.CaseStopIsLoweredTimerOff.ET;
GVL_CONVEYORS.GL8.CaseStop1LoweredSwitchIsOff := GVL_CONVEYORS.GL8.CaseStop1IsLoweredTimerOffDoneBit;

// DE-BOUNCE TIMER FOR GL8 CASE STOP1 IS RAISED SWITCH ON
GVL_CONVEYORS.GL8.CaseStop1IsRaisedTimerOn (IN := GVL_CONVEYORS.GL8.Case_Stop_Load_1_Extended_Right AND GVL_CONVEYORS.GL8.Case_Stop_Load_1_Extended_Left , PT := T#500MS);
GVL_CONVEYORS.GL8.CaseStop1IsRaisedTimerOnDoneBit := GVL_CONVEYORS.GL8.CaseStop1IsRaisedTimerOn.Q;
GVL_CONVEYORS.GL8.CaseStop1IsRaisedTimerOnElapsedTime := GVL_CONVEYORS.GL8.CaseStop1IsRaisedTimerOn.ET;
GVL_CONVEYORS.GL8.CaseStop1RaisedSwitchIsOn := GVL_CONVEYORS.GL8.CaseStop1IsRaisedTimerOnDoneBit;

// DE-BOUNCE TIMER FOR GL8 CASE STOP1 IS RAISED SWITCH OFF
GVL_CONVEYORS.GL8.CaseStop1IsRaisedTimerOff (IN := GVL_CONVEYORS.GL8.Case_Stop_Load_1_Extended_Right AND GVL_CONVEYORS.GL8.Case_Stop_Load_1_Extended_Left , PT := T#500MS);
GVL_CONVEYORS.GL8.CaseStop1IsRaisedTimerOffDoneBit := GVL_CONVEYORS.GL8.CaseStop1IsRaisedTimerOff.Q;
GVL_CONVEYORS.GL8.CaseStop1IsRaisedTimerOffElapsedTime := GVL_CONVEYORS.GL8.CaseStop1IsRaisedTimerOff.ET;
GVL_CONVEYORS.GL8.CaseStop1RaisedSwitchIsOff := GVL_CONVEYORS.GL8.CaseStop1IsRaisedTimerOffDoneBit;

// DE-BOUNCE TIMER FOR GL8 CASE STOP2 IS LOWERED SWITCH ON
GVL_CONVEYORS.GL8.CaseStop2IsLoweredTimerOn (IN := GVL_CONVEYORS.GL8.Case_Stop_Load_2_Retracted_Right AND GVL_CONVEYORS.GL8.Case_Stop_Load_2_Retracted_Left , PT := T#500MS);
GVL_CONVEYORS.GL8.CaseStop2IsLoweredTimerOnDoneBit := GVL_CONVEYORS.GL8.CaseStop2IsLoweredTimerOn.Q;
GVL_CONVEYORS.GL8.CaseStop2IsLoweredTimerOnElapsedTime := GVL_CONVEYORS.GL8.CaseStop2IsLoweredTimerOn.ET;
GVL_CONVEYORS.GL8.CaseStop2LoweredSwitchIsOn := GVL_CONVEYORS.GL8.CaseStop2IsLoweredTimerOnDoneBit;

// DE-BOUNCE TIMER FOR GL8 CASE STOP2 IS LOWERED SWITCH OFF
GVL_CONVEYORS.GL8.CaseStop2IsLoweredTimerOFF (IN := GVL_CONVEYORS.GL8.Case_Stop_Load_2_Retracted_Right AND GVL_CONVEYORS.GL8.Case_Stop_Load_2_Retracted_Left , PT := T#500MS);
GVL_CONVEYORS.GL8.CaseStopIsLoweredTimerOffDoneBit := GVL_CONVEYORS.GL8.CaseStop2IsLoweredTimerOff.Q;
GVL_CONVEYORS.GL8.CaseStop2IsLoweredTimerOffElapsedTime := GVL_CONVEYORS.GL8.CaseStop2IsLoweredTimerOff.ET;
GVL_CONVEYORS.GL8.CaseStop2LoweredSwitchIsOff := GVL_CONVEYORS.GL8.CaseStop2IsLoweredTimerOffDoneBit;

// DE-BOUNCE TIMER FOR GL8 CASE STOP2 IS RAISED SWITCH ON
GVL_CONVEYORS.GL8.CaseStop2IsRaisedTimerOn (IN := GVL_CONVEYORS.GL8.Case_Stop_Load_2_Extended_Right AND GVL_CONVEYORS.GL8.Case_Stop_Load_2_Extended_Left , PT := T#500MS);
GVL_CONVEYORS.GL8.CaseStop2IsRaisedTimerOnDoneBit := GVL_CONVEYORS.GL8.CaseStop2IsRaisedTimerOn.Q;
GVL_CONVEYORS.GL8.CaseStop2IsRaisedTimerOnElapsedTime := GVL_CONVEYORS.GL8.CaseStop2IsRaisedTimerOn.ET;
GVL_CONVEYORS.GL5B.CaseStopRaisedSwitchIsOn := GVL_CONVEYORS.GL5B.CaseStopIsRaisedTimerOnDoneBit;

